	4: ;(*kabinet*)
		IF fb_kl6301_0.GroupReceive.number <10 AND fb_kl6301_0.GroupReceive.number <>0 THEN kabinet_hvac.heat_mode:=fb_kl6301_0.GroupReceive.number;END_IF
		CASE fb_kl6301_0.GroupReceive.number OF
			0:		fb_temp_read(Group_Address:=kabinet_T_EIB_addr, strData_Rec:=fb_KL6301_0.str_Data_Rec, rData=>kabinet_HVAC.cur_t); (*temperature*)
			1:		fb_setpoint_read(Group_address:=kabinet_cooling_EIB_addr, strData_Rec:=fb_KL6301_0.str_Data_Rec, byData=>setpoint_kabinet_dpt4 ); (*cooling*)
					CASE REAL_TO_INT(setpoint_kabinet_dpt4*100/255.0) OF
						0..30:		kabinet_hvac.heat_speed:=1;
									kabinet_hvac.t_ust_cool:= REAL_TO_INT(setpoint_kabinet_dpt4*100/255.0); (*low speed*)
						31..59:		kabinet_hvac.heat_speed:=2;
									kabinet_hvac.t_ust_cool:= REAL_TO_INT(setpoint_kabinet_dpt4*100/255.0-30); (*med speed*)
						60..100:	kabinet_hvac.heat_speed:=3;
									kabinet_hvac.t_ust_cool:= REAL_TO_INT(setpoint_kabinet_dpt4*100/255.0-60); (*high speed*)
					END_CASE
					kabinet_hvac.cur_t_ust:=kabinet_hvac.t_ust_cool;
					(*fb_actual_setpoint_send(group_address:=kabinet_actual_setpoint_addr, str_Rec:=fb_kl6301_0.str_Data_Rec, rData:=kabinet_hvac.cur_t_ust);*)

			2:		fb_setpoint_read(Group_address:=kabinet_heating_EIB_addr, strData_Rec:=fb_KL6301_0.str_Data_Rec, byData=>setpoint_kabinet_dpt4 );  (*heating*)
					CASE REAL_TO_INT(setpoint_kabinet_dpt4*100/255.0) OF
						0..30:		kabinet_hvac.heat_speed:=1;
									kabinet_hvac.t_ust_heat:= REAL_TO_INT(setpoint_kabinet_dpt4*100/255.0); (*low speed*)
						31..59:		kabinet_hvac.heat_speed:=2;
									kabinet_hvac.t_ust_heat:= REAL_TO_INT(setpoint_kabinet_dpt4*100/255.0-30); (*med speed*)
						60..100:	kabinet_hvac.heat_speed:=3;
									kabinet_hvac.t_ust_heat:= REAL_TO_INT(setpoint_kabinet_dpt4*100/255.0-60); (*high speed*)
					END_CASE
					kabinet_hvac.cur_t_ust:=kabinet_hvac.t_ust_heat;
					(*fb_actual_setpoint_send(group_address:=kabinet_actual_setpoint_addr, str_Rec:=fb_kl6301_0.str_Data_Rec, rData:=kabinet_hvac.cur_t_ust);*)


			3:		fb_setpoint_read(Group_address:=kabinet_fan_EIB_addr, strData_Rec:=fb_KL6301_0.str_Data_Rec, byData=>fanspeed_dpt4);
					kabinet_HVAC.heat_speed:=REAL_TO_USINT(fanspeed_dpt4*100/255.0);
			4:		KABINET_HVAC.heat_mode:=0;
			5:		fb_actual_setpoint_read(Group_Address:=kabinet_actual_setpoint_addr, strData_Rec:=fb_KL6301_0.str_Data_Rec );
					kabinet_hvac.cur_t_ust:=fb_actual_setpoint_read.rData;

		END_CASE;

	5: ;(*dytjacha*)
		IF fb_kl6301_0.GroupReceive.number <10 AND fb_kl6301_0.GroupReceive.number <>0 THEN dytjacha_hvac.heat_mode:=fb_kl6301_0.GroupReceive.number;END_IF
		CASE fb_kl6301_0.GroupReceive.number OF
			0:		fb_temp_read(Group_Address:=dytjacha_T_EIB_addr, strData_Rec:=fb_KL6301_0.str_Data_Rec, rData=>dytjacha_HVAC.cur_t); (*temperature*)
			1:		fb_setpoint_read(Group_address:=dytjacha_cooling_EIB_addr, strData_Rec:=fb_KL6301_0.str_Data_Rec, byData=>setpoint_dytjacha_dpt4 ); (*cooling*)
					CASE REAL_TO_INT(setpoint_dytjacha_dpt4*100/255.0) OF
						0..30:		dytjacha_hvac.heat_speed:=1;
									dytjacha_hvac.t_ust_cool:= REAL_TO_INT(setpoint_dytjacha_dpt4*100/255.0); (*low speed*)
						31..59:		dytjacha_hvac.heat_speed:=2;
									dytjacha_hvac.t_ust_cool:= REAL_TO_INT(setpoint_dytjacha_dpt4*100/255.0-30); (*med speed*)
						60..100:	dytjacha_hvac.heat_speed:=3;
									dytjacha_hvac.t_ust_cool:= REAL_TO_INT(setpoint_dytjacha_dpt4*100/255.0-60); (*high speed*)
					END_CASE
					dytjacha_hvac.cur_t_ust:=dytjacha_hvac.t_ust_cool;
					(*fb_actual_setpoint_send(group_address:=dytjacha_actual_setpoint_addr, str_Rec:=fb_kl6301_0.str_Data_Rec, rData:=dytjacha_hvac.cur_t_ust);*)

			2:		fb_setpoint_read(Group_address:=dytjacha_heating_EIB_addr, strData_Rec:=fb_KL6301_0.str_Data_Rec, byData=>setpoint_dytjacha_dpt4 );  (*heating*)
					CASE REAL_TO_INT(setpoint_dytjacha_dpt4*100/255.0) OF
						0..30:		dytjacha_hvac.heat_speed:=1;
									dytjacha_hvac.t_ust_heat:= REAL_TO_INT(setpoint_dytjacha_dpt4*100/255.0); (*low speed*)
						31..59:		dytjacha_hvac.heat_speed:=2;
									dytjacha_hvac.t_ust_heat:= REAL_TO_INT(setpoint_dytjacha_dpt4*100/255.0-30); (*med speed*)
						60..100:	dytjacha_hvac.heat_speed:=3;
									dytjacha_hvac.t_ust_heat:= REAL_TO_INT(setpoint_dytjacha_dpt4*100/255.0-60); (*high speed*)
					END_CASE
					dytjacha_hvac.cur_t_ust:=dytjacha_hvac.t_ust_heat;
					(*fb_actual_setpoint_send(group_address:=dytjacha_actual_setpoint_addr, str_Rec:=fb_kl6301_0.str_Data_Rec, rData:=dytjacha_hvac.cur_t_ust);*)


			3:		fb_setpoint_read(Group_address:=dytjacha_fan_EIB_addr, strData_Rec:=fb_KL6301_0.str_Data_Rec, byData=>fanspeed_dpt4);
					dytjacha_HVAC.heat_speed:=REAL_TO_USINT(fanspeed_dpt4*100/255.0);
			4:		DYTJACHA_HVAC.heat_mode:=0;
			5:		fb_actual_setpoint_read(Group_Address:=dytjacha_actual_setpoint_addr, strData_Rec:=fb_KL6301_0.str_Data_Rec );
					dytjacha_hvac.cur_t_ust:=fb_actual_setpoint_read.rData;

		END_CASE;

	6: ;(*spalnya*)
		IF fb_kl6301_0.GroupReceive.number <10 AND fb_kl6301_0.GroupReceive.number <>0 THEN spalnya_hvac.heat_mode:=fb_kl6301_0.GroupReceive.number;END_IF
		CASE fb_kl6301_0.GroupReceive.number OF
			0:		fb_temp_read(Group_Address:=spalnya_T_EIB_addr, strData_Rec:=fb_KL6301_0.str_Data_Rec, rData=>spalnya_HVAC.cur_t); (*temperature*)
			1:		fb_setpoint_read(Group_address:=spalnya_cooling_EIB_addr, strData_Rec:=fb_KL6301_0.str_Data_Rec, byData=>setpoint_spalnya_dpt4 ); (*cooling*)
					CASE REAL_TO_INT(setpoint_spalnya_dpt4*100/255.0) OF
						0..30:		spalnya_hvac.heat_speed:=1;
									spalnya_hvac.t_ust_cool:= REAL_TO_INT(setpoint_spalnya_dpt4*100/255.0); (*low speed*)
						31..59:		spalnya_hvac.heat_speed:=2;
									spalnya_hvac.t_ust_cool:= REAL_TO_INT(setpoint_spalnya_dpt4*100/255.0-30); (*med speed*)
						60..100:	spalnya_hvac.heat_speed:=3;
									spalnya_hvac.t_ust_cool:= REAL_TO_INT(setpoint_spalnya_dpt4*100/255.0-60); (*high speed*)
					END_CASE
					spalnya_hvac.cur_t_ust:=spalnya_hvac.t_ust_cool;
					(*fb_actual_setpoint_send(group_address:=spalnya_actual_setpoint_addr, str_Rec:=fb_kl6301_0.str_Data_Rec, rData:=spalnya_hvac.cur_t_ust);*)

			2:		fb_setpoint_read(Group_address:=spalnya_heating_EIB_addr, strData_Rec:=fb_KL6301_0.str_Data_Rec, byData=>setpoint_spalnya_dpt4 );  (*heating*)
					CASE REAL_TO_INT(setpoint_spalnya_dpt4*100/255.0) OF
						0..30:		spalnya_hvac.heat_speed:=1;
									spalnya_hvac.t_ust_heat:= REAL_TO_INT(setpoint_spalnya_dpt4*100/255.0); (*low speed*)
						31..59:		spalnya_hvac.heat_speed:=2;
									spalnya_hvac.t_ust_heat:= REAL_TO_INT(setpoint_spalnya_dpt4*100/255.0-30); (*med speed*)
						60..100:	spalnya_hvac.heat_speed:=3;
									spalnya_hvac.t_ust_heat:= REAL_TO_INT(setpoint_spalnya_dpt4*100/255.0-60); (*high speed*)
					END_CASE
					spalnya_hvac.cur_t_ust:=spalnya_hvac.t_ust_heat;
					(*fb_actual_setpoint_send(group_address:=spalnya_actual_setpoint_addr, str_Rec:=fb_kl6301_0.str_Data_Rec, rData:=spalnya_hvac.cur_t_ust);*)


			3:		fb_setpoint_read(Group_address:=spalnya_fan_EIB_addr, strData_Rec:=fb_KL6301_0.str_Data_Rec, byData=>fanspeed_dpt4);
					spalnya_HVAC.heat_speed:=REAL_TO_USINT(fanspeed_dpt4*100/255.0);
			4:		SPALNYA_HVAC.heat_mode:=0;
			5:		fb_actual_setpoint_read(Group_Address:=spalnya_actual_setpoint_addr, strData_Rec:=fb_KL6301_0.str_Data_Rec );
					spalnya_hvac.cur_t_ust:=fb_actual_setpoint_read.rData;

		END_CASE;
END_CASE



(*hdl gate can transmit 2byte values, but they can not be assigned to DLP panel AC unit setpoint value directly,
so for every setpoint value in range [20,30] a 1 bit eib telegram with corresponding  adress +100 ( [120,130] ) should be generated and transmitted to HDL logic module and then
logic module assigns it to apropriate value DLP panel AC unit. 
amen*)
fb_setpoint_switch_send.iMode:=2;
fb_setpoint_switch_send.bStart:=TRUE;
IF vitalnya_hvac.cur_t_ust_prev <> vitalnya_hvac.cur_t_ust THEN
	fb_setpoint_switch_send.Group_Address.NUMBER:=REAL_TO_BYTE(vitalnya_hvac.cur_t_ust)+100;
	fb_setpoint_switch_send.Group_Address.MAIN:=1;
	fb_setpoint_switch_send.Group_Address.SUB_MAIN:=1;
	fb_setpoint_switch_send(str_Rec:=fb_KL6301_0.str_Data_Rec, bData:=FALSE);
	fb_setpoint_switch_send(str_Rec:=fb_KL6301_0.str_Data_Rec, bData:=TRUE);
END_IF
IF kino_hvac.cur_t_ust_prev <> kino_hvac.cur_t_ust THEN
	fb_setpoint_switch_send.Group_Address.NUMBER:=REAL_TO_BYTE(kino_hvac.cur_t_ust)+100;
	fb_setpoint_switch_send.Group_Address.MAIN:=1;
	fb_setpoint_switch_send.Group_Address.SUB_MAIN:=2;
	fb_setpoint_switch_send(str_Rec:=fb_KL6301_0.str_Data_Rec, bData:=1);
	fb_setpoint_switch_send(str_Rec:=fb_KL6301_0.str_Data_Rec, bData:=0);
END_IF
IF studio_hvac.cur_t_ust_prev <> studio_hvac.cur_t_ust THEN
	fb_setpoint_switch_send.Group_Address.NUMBER:=REAL_TO_BYTE(studio_hvac.cur_t_ust)+100;
	fb_setpoint_switch_send.Group_Address.MAIN:=1;
	fb_setpoint_switch_send.Group_Address.SUB_MAIN:=3;
	fb_setpoint_switch_send(str_Rec:=fb_KL6301_0.str_Data_Rec, bData:=1);
	fb_setpoint_switch_send(str_Rec:=fb_KL6301_0.str_Data_Rec, bData:=0);
END_IF
IF kabinet_hvac.cur_t_ust_prev <> kabinet_hvac.cur_t_ust THEN
	fb_setpoint_switch_send.Group_Address.NUMBER:=REAL_TO_BYTE(kabinet_hvac.cur_t_ust)+100;
	fb_setpoint_switch_send.Group_Address.MAIN:=1;
	fb_setpoint_switch_send.Group_Address.SUB_MAIN:=4;
	fb_setpoint_switch_send(str_Rec:=fb_KL6301_0.str_Data_Rec, bData:=1);
	fb_setpoint_switch_send(str_Rec:=fb_KL6301_0.str_Data_Rec, bData:=0);
END_IF
IF dytjacha_hvac.cur_t_ust_prev <> dytjacha_hvac.cur_t_ust THEN
	fb_setpoint_switch_send.Group_Address.NUMBER:=REAL_TO_BYTE(dytjacha_hvac.cur_t_ust)+100;
	fb_setpoint_switch_send.Group_Address.MAIN:=1;
	fb_setpoint_switch_send.Group_Address.SUB_MAIN:=5;
	fb_setpoint_switch_send(str_Rec:=fb_KL6301_0.str_Data_Rec, bData:=1);
	fb_setpoint_switch_send(str_Rec:=fb_KL6301_0.str_Data_Rec, bData:=0);
END_IF
IF spalnya_hvac.cur_t_ust_prev <> spalnya_hvac.cur_t_ust THEN
	fb_setpoint_switch_send.Group_Address.NUMBER:=REAL_TO_BYTE(spalnya_hvac.cur_t_ust)+100;
	fb_setpoint_switch_send.Group_Address.MAIN:=1;
	fb_setpoint_switch_send.Group_Address.SUB_MAIN:=6;
	fb_setpoint_switch_send(str_Rec:=fb_KL6301_0.str_Data_Rec, bData:=1);
	fb_setpoint_switch_send(str_Rec:=fb_KL6301_0.str_Data_Rec, bData:=0);
END_IF
END_ACTION
ACTION timers:
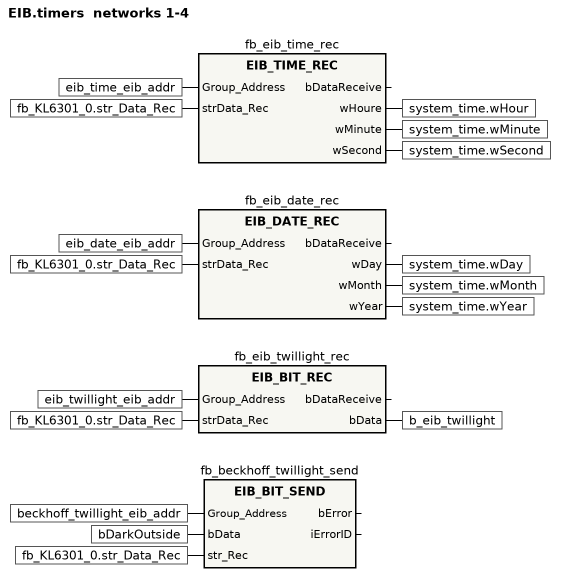
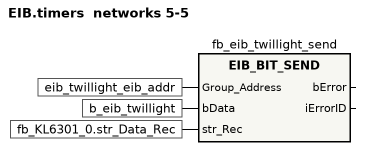
_FBD_ (* Function Block Diagram *)
NETWORK 1
	fb_eib_time_rec:EIB_TIME_REC(Group_Address: eib_time_eib_addr, strData_Rec: fb_KL6301_0.str_Data_Rec, wHoure => system_time.wHour, wMinute => system_time.wMinute, wSecond => system_time.wSecond)
NETWORK 2
	fb_eib_date_rec:EIB_DATE_REC(Group_Address: eib_date_eib_addr, strData_Rec: fb_KL6301_0.str_Data_Rec, wDay => system_time.wDay, wMonth => system_time.wMonth, wYear => system_time.wYear)
NETWORK 3
	fb_eib_twillight_rec:EIB_BIT_REC(Group_Address: eib_twillight_eib_addr, strData_Rec: fb_KL6301_0.str_Data_Rec, bData => b_eib_twillight)
NETWORK 4
	fb_beckhoff_twillight_send:EIB_BIT_SEND(Group_Address: beckhoff_twillight_eib_addr, bData: bDarkOutside, str_Rec: fb_KL6301_0.str_Data_Rec)
NETWORK 5
	fb_eib_twillight_send:EIB_BIT_SEND(Group_Address: eib_twillight_eib_addr, bData: b_eib_twillight, str_Rec: fb_KL6301_0.str_Data_Rec)
_END_FBD_
(* the same logic as Structured Text *)
(* Network 1 *)
fb_eib_time_rec(Group_Address := eib_time_eib_addr, strData_Rec := fb_KL6301_0.str_Data_Rec);
system_time.wHour := fb_eib_time_rec.wHoure;
system_time.wMinute := fb_eib_time_rec.wMinute;
system_time.wSecond := fb_eib_time_rec.wSecond;
(* Network 2 *)
fb_eib_date_rec(Group_Address := eib_date_eib_addr, strData_Rec := fb_KL6301_0.str_Data_Rec);
system_time.wDay := fb_eib_date_rec.wDay;
system_time.wMonth := fb_eib_date_rec.wMonth;
system_time.wYear := fb_eib_date_rec.wYear;
(* Network 3 *)
fb_eib_twillight_rec(Group_Address := eib_twillight_eib_addr, strData_Rec := fb_KL6301_0.str_Data_Rec);
b_eib_twillight := fb_eib_twillight_rec.bData;
(* Network 4 *)
fb_beckhoff_twillight_send(Group_Address := beckhoff_twillight_eib_addr, bData := bDarkOutside, str_Rec := fb_KL6301_0.str_Data_Rec);
(* Network 5 *)
fb_eib_twillight_send(Group_Address := eib_twillight_eib_addr, bData := b_eib_twillight, str_Rec := fb_KL6301_0.str_Data_Rec);
END_ACTION

(* POU RANGE_TO_RANGE, ST *)
FUNCTION RANGE_TO_RANGE : INT
VAR_INPUT
	by_input:BYTE;
	in_low_value: INT;
	in_high_value:INT;
	out_low_value: INT;
	out_high_value:INT;
END_VAR
VAR
	r_res: REAL;
	r_input: REAL;
END_VAR
r_input:=BYTE_TO_REAL(by_input);
IF out_high_value>out_low_value THEN
	r_res:=r_input/(in_high_value - in_low_value)*(out_high_value - out_low_value);
ELSE
	r_res:=out_low_value - (r_input / (in_high_value - in_low_value)*(out_low_value - out_high_value));
END_IF
RANGE_TO_RANGE:=REAL_TO_INT(r_res);
END_FUNCTION

(* POU GREATEST_OF, ST *)
FUNCTION GREATEST_OF : REAL
VAR_INPUT
	r_in1,r_in2:REAL;
END_VAR
VAR
END_VAR
IF r_in1>=r_in2 THEN
	GREATEST_OF:=r_in1;
ELSE
	GREATEST_OF:=r_in2;
END_IF
END_FUNCTION

(* POU LIGHT, ST *)
PROGRAM LIGHT
VAR
	tambur1, tambur2,tambur3 : SWITCH;
	korydor : SWITCH;
	spalnya1,spalnya2, spalnya_balk:SWITCH;
	dytjacha1,dytjacha2  : SWITCH;
	su1 : SWITCH;
	su2: SWITCH;
	garderob1, garderob2 : SWITCH;

	tLightWindow: TIME;		(*Час, який світло світиться після спрацювання сенсора руху*)

	VENT_TIMER: TOF;		(*Таймер роботи вентилятора в пустому туалеті*)
	vent_timer_start: R_TRIG;
	test: BOOL;

	CHOVEN_TIMER: TOF;	(*Таймер роботи світильника на човні*)

	bChovenTimerOverride: SEMA;		(*Перевага вимикача над таймером*)
	bGarderobTimerOverride: SEMA;		(*Перевага вимикача над таймером*)
	KORYDOR_TIMER: TOF;		(*Таймер роботи світла в коридорі*)
	KORYDOR_F: F_TRIG;
	GARDEROB_TIMER: TOF;		(*Таймер роботи світла в гардеробі*)
	GARDEROB_F: F_TRIG;		(*Спрацювання сенсора руху в гардеробі*)
	KORYDOR_SEMA:SEMA;
	su_light: BOOL;
	vymykach3: BOOL;

	fb_light_write:EIB_BIT_SEND;
	block_korydor, block_garderob, block_choven: BOOL;

END_VAR
tLightWindow:=t#60s;

IF fb_moove_sensors_read.bData THEN
	moove_sensors:=(*bDarkOutside*)TRUE;
ELSE
	moove_sensors:=FALSE;
END_IF

(*Опитування вимикачів*)
tambur1(IN:=sw_tambur1);
tambur2(IN:=sw_tambur3_2);
tambur3(IN:=sw_tambur3);



spalnya1(IN:=sw_spalnya1 XOR sw_spalnya4);
spalnya2(IN:=sw_spalnya2 XOR sw_spalnya3);
spalnya_balk(IN:=sw_spalnya_balk);

dytjacha1(IN:=sw_dytjacha1);
dytjacha2(IN:=sw_dytjacha2);

su1(IN:=sw_su1);
su2(IN:=sw_su2);




(*запуск вечірніх таймерів світла*)





(*обробка сигналів вимикачів та таймерів*)
IF fb_bar_read.bDataReceive THEN
	IF tambur1.short THEN bar:= NOT bar; END_IF
ELSE
	bar:=fb_bar_read.bData;
END_IF

(*Відправка на 1,2 поверхи значення вимикача*)
data2floor[6].0:=sw_tambur3_2;
data1floor[2].1:=sw_tambur3_2;

CHOVEN_TIMER(IN:= NOT fb_choven_read.bData AND NOT moove_skhody, PT:= tLightWindow);
IF fb_choven_read.bData THEN
	choven:=TRUE;
ELSE
	IF moove_sensors  AND  CHOVEN_timer.Q	THEN  choven:=TRUE;
	ELSE
	choven:=FALSE;
	END_IF
END_IF


korydor(IN:=sw_korydor);
KORYDOR_TIMER(IN:=  NOT fb_korydor_lampa_read.bData  AND NOT moove_korydor, PT:= tLightWindow);

IF fb_korydor_lampa_read.bData THEN
	korydor_lampa:=TRUE;
ELSE
		korydor_lampa:=KORYDOR_TIMER.Q;
END_IF

IF fb_korydor_skeli_read.bData THEN
	korydor_skeli:=TRUE;
ELSE
	korydor_skeli:=KORYDOR_TIMER.Q;
END_IF

IF fb_korydor_svitlo_read.bDataReceive THEN
	KORYDOR_F(clk:=korydor_timer.Q);
	KORYDOR_SEMA(CLAIM:=(NOT korydor_svitlo AND korydor.short ), RELEASE:=(korydor_svitlo AND korydor.short) OR KORYDOR_f.Q);
	korydor_svitlo:=KORYDOR_SEMA.BUSY;
ELSE
	korydor_svitlo:= fb_korydor_svitlo_read.bData;

END_IF

IF fb_spalnya_kulbaba_read.bDataReceive THEN
	IF spalnya1.short THEN spalnya_kulbaba:=NOT spalnya_kulbaba; END_IF
ELSE
	spalnya_kulbaba:=fb_spalnya_kulbaba_read.bData;
END_IF

IF fb_spalnya_kontrazhur_read.bDataReceive XOR fb_spalnya_kontrazhur_b_read.bDataReceive  XOR fb_spalnya_kontrazhur_l_read.bDataReceive  THEN
	IF spalnya2.short THEN
		 spalnya_kontrazhur:= NOT spalnya_kontrazhur;
		spalnya_kontrazhur_b:=spalnya_kontrazhur;
		spalnya_kontrazhur_l:=spalnya_kontrazhur;
 	END_IF
ELSE
	IF NOT fb_spalnya_kontrazhur_read.bDataReceive THEN spalnya_kontrazhur:= fb_spalnya_kontrazhur_read.bData; END_IF
	IF NOT fb_spalnya_kontrazhur_l_read.bDataReceive THEN spalnya_kontrazhur_l:= fb_spalnya_kontrazhur_l_read.bData; END_IF
	IF NOT fb_spalnya_kontrazhur_b_read.bDataReceive THEN spalnya_kontrazhur_b:= fb_spalnya_kontrazhur_b_read.bData; END_IF
END_IF

IF fb_spalnya_balkon_read.bDataReceive THEN
	IF  spalnya_balk.short  THEN spalnya_balkon:=NOT spalnya_balkon; END_IF
ELSE
	spalnya_balkon:=fb_spalnya_balkon_read.bData;
END_IF

IF fb_dytjacha_read.bDataReceive THEN
	IF dytjacha1.short THEN dytjacha:= NOT dytjacha; END_IF
ELSE
	dytjacha:=fb_dytjacha_read.bData;
END_IF

IF fb_dytjacha_bra_read.bDataReceive THEN
	IF dytjacha2.short THEN dytjacha_bra:= NOT dytjacha_bra; END_IF
ELSE
	dytjacha_bra:=fb_dytjacha_bra_read.bData;
END_IF


IF fb_su3_stina_read.bDataReceive AND  fb_su3_kontrazhur_k_read.bDataReceive THEN
	IF su2.short THEN
		su3_stina:= NOT su3_stina;
		(*su3_kontrazhur_k:= su3_stina; *)
	END_IF
ELSE
	IF NOT fb_su3_stina_read.bDataReceive THEN
		 su3_stina:=fb_su3_stina_read.bData;
	END_IF
	IF NOT fb_su3_kontrazhur_k_read.bDataReceive THEN
		su3_kontrazhur_k:= fb_su3_kontrazhur_k_read.bData;
	END_IF
END_IF



IF fb_su3_bra_read.bDataReceive XOR fb_su3_lampa_read.bDataReceive XOR fb_su3_kontrazhur_read.bDataReceive THEN
	IF su2.long THEN
		su3_bra:= NOT su3_bra;
		su3_lampa:= su3_bra;
		su3_kontrazhur:=su3_lampa;
	END_IF
ELSE
	IF NOT  fb_su3_bra_read.bDataReceive THEN su3_bra:= fb_su3_bra_read.bData;END_IF
	IF NOT fb_su3_lampa_read.bDataReceive THEN su3_lampa:=fb_su3_lampa_read.bData; END_IF
	IF NOT  fb_su3_kontrazhur_read.bDataReceive THEN su3_kontrazhur:=fb_su3_kontrazhur_read.bData; END_IF
END_IF

IF su1.long THEN su3_vent:= NOT su3_vent; END_IF

IF fb_su3_pidsvitka_read.bDataReceive THEN
	IF su1.short THEN su3_pidsvitka:= NOT su3_pidsvitka; END_IF
ELSE
	su3_pidsvitka:=fb_su3_pidsvitka_read.bData;
END_IF

(*IF su1.short AND NOT su3_vent THEN su3_vent:=TRUE; END_IF; *) (*вмикання вентилятора разом зі світлом*)

(*
вмикання вентилятора на деякий час після того, як вимикається все світло у ванній

su_light:=su3_stina OR su3_kontrazhur OR su3_bra OR su3_pidsvitka;

vent_timer_start(CLK:=NOT su_light );
VENT_TIMER(PT:=tOffDelay,IN:=vent_timer_start.Q);
IF NOT su_light THEN
	su3_vent:= VENT_TIMER.Q;
END_IF
*)


garderob1(IN:=sw_garderob1);
garderob2(IN:=sw_garderob2);
GARDEROB_F(CLK:=moove_garderob);
GARDEROB_TIMER(IN:= GARDEROB_F.Q, PT:= tLightWindow*2);

IF fb_serverna_read.bDataReceive THEN
	IF garderob2.short THEN serverna := NOT serverna; END_IF
ELSE
	Serverna:=fb_serverna_read.bData;
END_IF

IF fb_garderob_read.bDataReceive THEN
(*	bGarderobTimerOverride(CLAIM:=  (NOT moove_garderob OR (NOT garderob AND garderob1.short)), RELEASE:=  (garderob AND  garderob1.short) );
	garderob:=bGarderobTimerOverride.BUSY;*)
	IF garderob1.short THEN garderob:= NOT garderob; END_IF
ELSE
	garderob:=fb_garderob_read.bData;
END_IF
END_PROGRAM

(* POU Vymykachi/SWITCH, ST *)
FUNCTION_BLOCK SWITCH
VAR_INPUT
	IN:BOOL;
	SHORT_OFF_DELAY, LONG_OFF_DELAY: TIME; (*час затримки вимкнення по короткому та довгому натисненню*)
END_VAR
VAR_OUTPUT
	short, long:BOOL;
END_VAR
VAR
	tChas: TIME; (*час доки кнопка натиснена*)
	TIMER: TON; (*таймер час натискання*)
	bPressed:BOOL;
	turn_off_long: BOOL;
	start_l, start_s:BOOL;
	bStan: BOOL:=FALSE;
END_VAR
short:=FALSE;
long:=FALSE;
TIMER(IN:=IN AND bStan, PT:=t#10s);
IF IN AND bStan THEN
	tChas:=timer.ET;
	bPressed:=TRUE;
ELSE
	bPressed:=FALSE;
END_IF;

IF NOT IN AND NOT bStan THEN
	tChas:=t#0ms;
END_IF;

IF bStan AND NOT IN THEN
	IF tChas <tLongPress THEN
		short:=TRUE;
	END_IF;
	IF tChas>=tLongPress THEN
		long:=TRUE;
	END_IF;
END_IF;
bStan := IN;
END_FUNCTION_BLOCK

(* POU shtory, ST *)
PROGRAM shtory
VAR
	inc1, inc: UINT;
	impulse: BOOL;
	last_move: UINT;
	impulse1: BOOL;
	last_move1: UINT;
	lift_move_dir, lift_move: BOOL;
	rising1: BOOL;
	falling1: BOOL;
	rising2: BOOL;
	falling2: BOOL;
	panel_shtory_move, panel_tul_move, panel_lift_move:BOOL;

	(*таймери для формування керуючих імпульсів*)
	timer_shtory_move, timer_shtory_stop,timer_tul_move, timer_tul_stop, move_lift_up, move_lift_down: TP;
	counter:CTU;
	shtory_move: BOOL;
	tul_move: BOOL;
	bBlock:BOOL;
	darkness_shtory_move: TP;
	btest: BOOL;

	eib_spalnya_shtory_status_send: EIB_BIT_SEND;
	eib_spalnya_tul_status_send: EIB_BIT_SEND;
	spalnya_shtory_status: BOOL;
	spalnya_tul_status: BOOL;
END_VAR
bBlock:=FALSE;
IF MAIN.fbRTC.stSystemTime.wHour=11 AND MAIN.fbRTC.stSystemTime.wMinute=0 AND MAIN.fbRTC.stSystemTime.wSecond<22 THEN
	bBlock:=TRUE;
	lift_down:=TRUE;
	lift_up:=FALSE;
	lift_move_dir:=FALSE;
	shtory_open:=TRUE;
	shtory_close:=FALSE;
	tul_open:=FALSE;
	tul_close:=TRUE;

ELSE
	(*детекція відсутності фронтів*)
	IF LIGHT.spalnya1.long = impulse THEN
		rising1:=0;
		falling1:=0;
	END_IF;

	IF LIGHT.spalnya2.long = impulse1  THEN
		rising2:=0;
		falling2:=0;
	END_IF;

	(*якщо клавіші довго  натиснені одночасно, то рухати ліфт, якщо довго і окремо - штори*)
	IF ( (LIGHT.spalnya1.long AND LIGHT.spalnya2.long) OR panel_lift_move)  AND NOT( move_lift_up.Q OR  move_lift_down.Q)  THEN
		lift_move:=1;
		lift_move_dir:= NOT lift_move_dir;
	ELSE

		(*ловим передній фронт довгого натискання першої клавіші*)
		IF LIGHT.spalnya1.long AND NOT impulse  AND NOT LIGHT.spalnya2.long THEN
			rising1:=1;
			falling1:=0;
		END_IF;

		(*задній фронт*)
		IF NOT LIGHT.spalnya1.long AND  impulse AND NOT LIGHT.spalnya2.long  THEN
			falling1:=1;
			rising1:=0;
		END_IF;

		(*ловим передній фронт довгого натискання другої клавіші*)
		IF LIGHT.spalnya2.long AND NOT impulse1 AND NOT LIGHT.spalnya1.long  THEN
			rising2:=1;
			falling2:=0;
		END_IF;

		(*ловим задній фронт довгого натискання другої клавіші*)
		IF NOT LIGHT.spalnya2.long AND  impulse1 AND NOT LIGHT.spalnya1.long THEN
			falling2:=1;
			rising2:=0;
		END_IF
	END_IF
	(*команди шторам та ліфту з панелей смартбаса*)
	eib_shtory(Group_Address:=shtory_spalnya_EIB_addr, strData_Rec:=fb_KL6301_0.str_Data_Rec);
	eib_tul(Group_Address:=tul_spalnya_EIB_addr, strData_Rec:=fb_KL6301_0.str_Data_Rec);
	eib_lift(Group_Address:=lift_spalnya_EIB_addr, strData_Rec:=fb_KL6301_0.str_Data_Rec);


	IF NOT eib_shtory_kabinet.bDataReceive THEN data2floor[7].0:=eib_shtory_kabinet.bData; END_IF
	IF NOT eib_tul_kabinet.bDataReceive THEN data2floor[7].1:=eib_tul_kabinet.bData; END_IF
	IF NOT eib_shtory_kino.bDataReceive THEN data2floor[7].2:=eib_shtory_kino.bData; END_IF
	IF NOT eib_tul_kino.bDataReceive THEN data2floor[7].3:=eib_tul_kino.bData; END_IF

	panel_tul_move:= NOT eib_tul.bDataReceive;
	panel_shtory_move:= NOT eib_shtory.bDataReceive;
	panel_lift_move:=NOT eib_lift.bDataReceive;


	shtory_move:= LIGHT.spalnya1.long OR panel_shtory_move;
	tul_move:= LIGHT.spalnya2.long OR panel_tul_move;



	(*формування імпульсів для керування шторами, тюлями та ліфтом*)
	timer_shtory_move(IN:=shtory_move, PT:=t#500ms);
	timer_shtory_stop(IN:=shtory_move , PT:=t#500ms);
	timer_tul_move(IN:=tul_move  , PT:=t#500ms);
	timer_tul_stop(IN:=tul_move , PT:=t#500ms);

	move_lift_up(IN:=lift_move AND lift_move_dir , PT:=t#20s,Q=>lift_up);
	move_lift_down(IN:=lift_move AND NOT lift_move_dir, PT:=t#20s, Q=>lift_down);



	darkness_shtory_move(IN:=bDarkOutside, PT:=t#15s);
	IF darkness_shtory_move.Q THEN
		shtory_open:=FALSE;
		shtory_close:=TRUE;
		tul_open:=FALSE;
		tul_close:=TRUE;
		bBlock:=TRUE;
	END_IF


	IF NOT bBlock THEN
		IF NOT (LIGHT.spalnya1.long AND LIGHT.spalnya2.long) THEN (*якщо не засік довгого затискання двох клавіш (ліфт не рухається) - рухати штори *)

		(*вибір рухати чи зупинити  штори*)
			IF shtory_move   THEN
				inc:=inc+1;
			END_IF;
			IF inc>2 THEN inc:=1; END_IF;

			(*вибір рухати чи зупинити  тюль*)
			IF tul_move THEN
				inc1:=inc1+1;
			END_IF;
			IF inc1>2 THEN inc1:=1; END_IF;

			CASE inc OF

				1:
				shtory_open:=timer_shtory_move.Q; (*відкривати*)
				shtory_close:= 0;
				last_move:=inc;
				spalnya_shtory_status:=1;

				2:
				shtory_close:=timer_shtory_move.Q;(*закривати*)
				shtory_open:= 0;
				last_move:=inc;
				spalnya_shtory_status:=0;

			END_CASE;

			CASE inc1 OF

				1:
				tul_open:=timer_tul_move.Q; (*відкривати*)
				tul_close:= 0;
				last_move1:=inc;
				spalnya_tul_status:=1;
				2:
				tul_close:=timer_tul_move.Q;(*закривати*)
				tul_open:= 0;
				last_move1:=inc;
				spalnya_tul_status:=0;
			END_CASE;

		END_IF;
	END_IF

	(*запам'ятовування стану довгого натискання для детекції фронтів*)

	impulse:=LIGHT.spalnya1.long;
	impulse1:=LIGHT.spalnya2.long;

	 lift_move:= 0;
END_IF
eib_status_send;

new_shtory;
END_PROGRAM
ACTION eib_status_send:
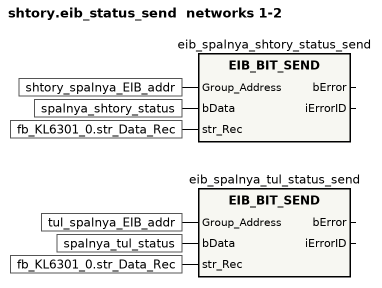
_FBD_ (* Function Block Diagram *)
NETWORK 1
	eib_spalnya_shtory_status_send:EIB_BIT_SEND(Group_Address: shtory_spalnya_EIB_addr, bData: spalnya_shtory_status, str_Rec: fb_KL6301_0.str_Data_Rec)
NETWORK 2
	eib_spalnya_tul_status_send:EIB_BIT_SEND(Group_Address: tul_spalnya_EIB_addr, bData: spalnya_tul_status, str_Rec: fb_KL6301_0.str_Data_Rec)
_END_FBD_
(* the same logic as Structured Text *)
(* Network 1 *)
eib_spalnya_shtory_status_send(Group_Address := shtory_spalnya_EIB_addr, bData := spalnya_shtory_status, str_Rec := fb_KL6301_0.str_Data_Rec);
(* Network 2 *)
eib_spalnya_tul_status_send(Group_Address := tul_spalnya_EIB_addr, bData := spalnya_tul_status, str_Rec := fb_KL6301_0.str_Data_Rec);
END_ACTION

(* POU new_shtory, CFC *)
PROGRAM new_shtory
VAR

END_VAR
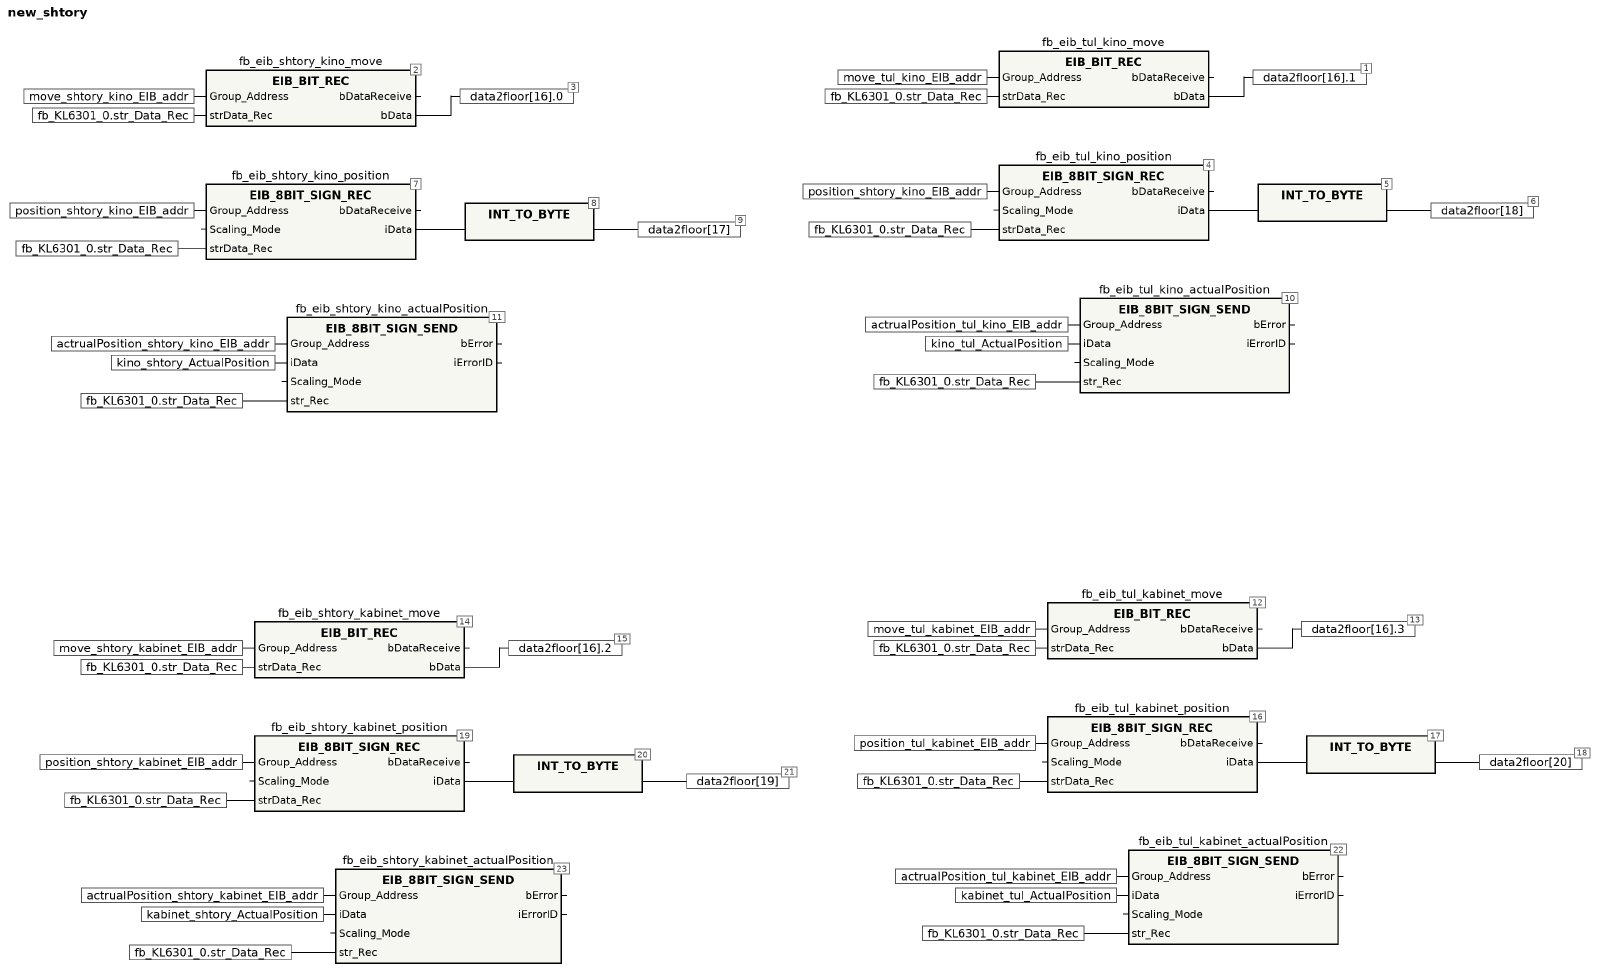
_CFC_ (* Continuous Function Chart, elements in execution order *)
#0 fb_eib_tul_kino_move:EIB_BIT_REC(Group_Address: move_tul_kino_EIB_addr, strData_Rec: fb_KL6301_0.str_Data_Rec)
#1 data2floor[16].1 <= #0.bData
#2 fb_eib_shtory_kino_move:EIB_BIT_REC(Group_Address: move_shtory_kino_EIB_addr, strData_Rec: fb_KL6301_0.str_Data_Rec)
#3 data2floor[16].0 <= #2.bData
#4 fb_eib_tul_kino_position:EIB_8BIT_SIGN_REC(Group_Address: position_shtory_kino_EIB_addr, Scaling_Mode: -, strData_Rec: fb_KL6301_0.str_Data_Rec)
#5 INT_TO_BYTE(#4.iData)
#6 data2floor[18] <= #5
#7 fb_eib_shtory_kino_position:EIB_8BIT_SIGN_REC(Group_Address: position_shtory_kino_EIB_addr, Scaling_Mode: -, strData_Rec: fb_KL6301_0.str_Data_Rec)
#8 INT_TO_BYTE(#7.iData)
#9 data2floor[17] <= #8
#10 fb_eib_tul_kino_actualPosition:EIB_8BIT_SIGN_SEND(Group_Address: actrualPosition_tul_kino_EIB_addr, iData: kino_tul_ActualPosition, Scaling_Mode: -, str_Rec: fb_KL6301_0.str_Data_Rec)
#11 fb_eib_shtory_kino_actualPosition:EIB_8BIT_SIGN_SEND(Group_Address: actrualPosition_shtory_kino_EIB_addr, iData: kino_shtory_ActualPosition, Scaling_Mode: -, str_Rec: fb_KL6301_0.str_Data_Rec)
#12 fb_eib_tul_kabinet_move:EIB_BIT_REC(Group_Address: move_tul_kabinet_EIB_addr, strData_Rec: fb_KL6301_0.str_Data_Rec)
#13 data2floor[16].3 <= #12.bData
#14 fb_eib_shtory_kabinet_move:EIB_BIT_REC(Group_Address: move_shtory_kabinet_EIB_addr, strData_Rec: fb_KL6301_0.str_Data_Rec)
#15 data2floor[16].2 <= #14.bData
#16 fb_eib_tul_kabinet_position:EIB_8BIT_SIGN_REC(Group_Address: position_tul_kabinet_EIB_addr, Scaling_Mode: -, strData_Rec: fb_KL6301_0.str_Data_Rec)
#17 INT_TO_BYTE(#16.iData)
#18 data2floor[20] <= #17
#19 fb_eib_shtory_kabinet_position:EIB_8BIT_SIGN_REC(Group_Address: position_shtory_kabinet_EIB_addr, Scaling_Mode: -, strData_Rec: fb_KL6301_0.str_Data_Rec)
#20 INT_TO_BYTE(#19.iData)
#21 data2floor[19] <= #20
#22 fb_eib_tul_kabinet_actualPosition:EIB_8BIT_SIGN_SEND(Group_Address: actrualPosition_tul_kabinet_EIB_addr, iData: kabinet_tul_ActualPosition, Scaling_Mode: -, str_Rec: fb_KL6301_0.str_Data_Rec)
#23 fb_eib_shtory_kabinet_actualPosition:EIB_8BIT_SIGN_SEND(Group_Address: actrualPosition_shtory_kabinet_EIB_addr, iData: kabinet_shtory_ActualPosition, Scaling_Mode: -, str_Rec: fb_KL6301_0.str_Data_Rec)
_END_CFC_
(* the same logic as Structured Text *)
fb_eib_tul_kino_move(Group_Address := move_tul_kino_EIB_addr, strData_Rec := fb_KL6301_0.str_Data_Rec);
data2floor[16].1 := fb_eib_tul_kino_move.bData;
fb_eib_shtory_kino_move(Group_Address := move_shtory_kino_EIB_addr, strData_Rec := fb_KL6301_0.str_Data_Rec);
data2floor[16].0 := fb_eib_shtory_kino_move.bData;
fb_eib_tul_kino_position(Group_Address := position_shtory_kino_EIB_addr, strData_Rec := fb_KL6301_0.str_Data_Rec);
data2floor[18] := INT_TO_BYTE(fb_eib_tul_kino_position.iData);
fb_eib_shtory_kino_position(Group_Address := position_shtory_kino_EIB_addr, strData_Rec := fb_KL6301_0.str_Data_Rec);
data2floor[17] := INT_TO_BYTE(fb_eib_shtory_kino_position.iData);
fb_eib_tul_kino_actualPosition(Group_Address := actrualPosition_tul_kino_EIB_addr, iData := kino_tul_ActualPosition, str_Rec := fb_KL6301_0.str_Data_Rec);
fb_eib_shtory_kino_actualPosition(Group_Address := actrualPosition_shtory_kino_EIB_addr, iData := kino_shtory_ActualPosition, str_Rec := fb_KL6301_0.str_Data_Rec);
fb_eib_tul_kabinet_move(Group_Address := move_tul_kabinet_EIB_addr, strData_Rec := fb_KL6301_0.str_Data_Rec);
data2floor[16].3 := fb_eib_tul_kabinet_move.bData;
fb_eib_shtory_kabinet_move(Group_Address := move_shtory_kabinet_EIB_addr, strData_Rec := fb_KL6301_0.str_Data_Rec);
data2floor[16].2 := fb_eib_shtory_kabinet_move.bData;
fb_eib_tul_kabinet_position(Group_Address := position_tul_kabinet_EIB_addr, strData_Rec := fb_KL6301_0.str_Data_Rec);
data2floor[20] := INT_TO_BYTE(fb_eib_tul_kabinet_position.iData);
fb_eib_shtory_kabinet_position(Group_Address := position_shtory_kabinet_EIB_addr, strData_Rec := fb_KL6301_0.str_Data_Rec);
data2floor[19] := INT_TO_BYTE(fb_eib_shtory_kabinet_position.iData);
fb_eib_tul_kabinet_actualPosition(Group_Address := actrualPosition_tul_kabinet_EIB_addr, iData := kabinet_tul_ActualPosition, str_Rec := fb_KL6301_0.str_Data_Rec);
fb_eib_shtory_kabinet_actualPosition(Group_Address := actrualPosition_shtory_kabinet_EIB_addr, iData := kabinet_shtory_ActualPosition, str_Rec := fb_KL6301_0.str_Data_Rec);
END_PROGRAM

(* POU HVAC/climate, ST *)
PROGRAM climate
VAR PERSISTENT

	t_out_avg_day, t_out_avg_10day:REAL;
	measures_this_day, meashured_days:INT;
	day_sum, ten_day_sum:REAL;
END_VAR


VAR

	t_tambur: REAL;
	t_su: REAL;
	t_spalnya : REAL;
	(*мінімум та максимум температур теплих підлог*)
	t_max: REAL;
	t_min: REAL;

	i: INT:=0;
	OAT_filter: 			FB_PT1;
	(*sensor filters*)
	t_tambur_filter: 		FB_PT1;
	t_su_filter : 			FB_PT1;
	t_spalnya_filter: 		FB_PT1;

	temperatureFiltersCycleTime:	TIME:=t#28ms;
	temperaturesFilterT1:			TIME:=t#60s;




END_VAR
(*фільтри показань сенсорів температури*)

OAT_filter.tCycletime:=temperatureFiltersCycleTime;
OAT_filter.tT1:=temperaturesFilterT1;
OAT_filter(fIn:=INT_TO_REAL(iT_out)/10, fOut=>t_out);

t_tambur_filter.tCycletime:=temperatureFiltersCycleTime;
t_tambur_filter.tT1:=temperaturesFilterT1;
t_tambur_filter (fIn:=INT_TO_REAL(iT_tambur)/10, fOut=>t_tambur);

t_su_filter.tCycletime:=temperatureFiltersCycleTime;
t_su_filter.tT1:=temperaturesFilterT1;
t_su_filter(fIn:=INT_TO_REAL(iT_su)/10, fOut=>t_su);

t_spalnya_filter.tCycletime:=temperatureFiltersCycleTime;
t_spalnya_filter.tT1:=temperaturesFilterT1;
t_spalnya_filter(fIn:=INT_TO_REAL(iT_spalnya)/10, fOut=>t_spalnya);


(*CASE MAIN.fbRTC.stSystemTime.wSecond OF*)



(*summer; *)

t_max:=70;
t_min:=20;
IF t_out<15 THEN

	IF t_tambur > t_max THEN (*вимкнути колектор, якщо підлога тепліша за верхню межу температури*)
		freshbar_col:=FALSE;
	ELSE
		IF t_tambur< t_min THEN (*увімкнути колектор, якщо підлога холодніша за нижню межу*)
			freshbar_col:=TRUE;
		ELSE
			freshbar_col:= FALSE; (*ПОСТАВИТИ В ЗАЛЕЖНІСТЬ ВІД ЗОВНІШНЬОЇ ТЕМПЕРАТУРИ*)
		END_IF
	END_IF

	IF t_su > t_max THEN
		su_col_pidloga:=FALSE;
		su_col_stina:=FALSE;
			serverna_col:=FALSE;
	ELSE
		IF t_su< t_min THEN
			su_col_pidloga:=TRUE;
			su_col_stina:=TRUE;
			serverna_col:=TRUE;
		ELSE
			su_col_pidloga:=FALSE; (*ПОСТАВИТИ В ЗАЛЕЖНІСТЬ ВІД ЗОВНІШНЬОЇ ТЕМПЕРАТУРИ*)
			su_col_stina:=FALSE;
			serverna_col:=FALSE;
		END_IF
	END_IF

	IF t_spalnya>t_max THEN (*щоб не вистигала підлога*)
		spalnya_col:=FALSE;
	ELSE
		IF t_spalnya<t_min THEN
			spalnya_col:=TRUE;
		ELSE
			spalnya_col:=SPALNYA_HVAC.tepla_pidloga;
		END_IF
	END_IF


END_IF

(*

IF VITALNYA_HVAC.heat_mode=0 THEN
				VITALNYA_HVAC.fancoil_speed:=0;
				(*VITALNYA_HVAC.collector:=2#00000000; all closed*)
				VITALNYA_HVAC.klapan:=16#7FFF;(*full closed*)
				VITALNYA_HVAC.zaslinka:=TRUE;(*closed*)
	END_IF

	IF KINO_HVAC.heat_mode=0 THEN
				KINO_HVAC.fancoil_speed:=0;
				(*KINO_HVAC.collector:=2#00000000; all closed*)
				KINO_HVAC.klapan:=16#7FFF;(*full closed*)
				KINO_HVAC.zaslinka:=TRUE;(*closed*)
	END_IF

	IF STUDIO_HVAC.heat_mode=0 THEN
				STUDIO_HVAC.fancoil_speed:=0;
				(*STUDIO_HVAC.collector:=2#00000000; all closed*)
				STUDIO_HVAC.klapan:=16#7FFF;(*full closed*)
				STUDIO_HVAC.zaslinka:=TRUE;(*closed*)
	END_IF

	IF KABINET_HVAC.heat_mode=0 THEN
				KABINET_HVAC.fancoil_speed:=0;
				(*KABINET_HVAC.collector:=2#00000000; all closed*)
				KABINET_HVAC.klapan:=16#7FFF;(*full closed*)
				KABINET_HVAC.zaslinka:=TRUE;(*closed*)
	END_IF

	IF DYTJACHA_HVAC.heat_mode=0 THEN
				DYTJACHA_HVAC.fancoil_speed:=0;
				(*DYTJACHA_HVAC.collector:=2#00000000; all closed*)
				DYTJACHA_HVAC.klapan:=16#7FFF;(*full closed*)
				DYTJACHA_HVAC.zaslinka:=TRUE;(*closed*)
	END_IF

	IF SPALNYA_HVAC.heat_mode=0 THEN
				SPALNYA_HVAC.fancoil_speed:=0;
				(*SPALNYA_HVAC.collector:=2#00000000; all closed*)
				SPALNYA_HVAC.klapan:=16#7FFF;(*full closed*)
				SPALNYA_HVAC.zaslinka:=TRUE;(*closed*)
	END_IF
*)





(*локальні змінні для фенкойлів 3го поверхну об'явлені в області виходів*)

(*------------------------fancoil speed --------------------------------------------------*)
IF EIB.fb_vitalnya_damper_ctrl_rec.bData THEN
	vitalnya_hvac.fancoil_speed:=1;
ELSE
	IF vitalnya_HVAC.heating_signal = 0  THEN
		CASE vitalnya_hvac.fancoil_speed OF
			0:	IF vitalnya_hvac.cooling_signal>0 THEN vitalnya_HVAC.fancoil_speed:=1; END_IF

			1:	IF vitalnya_hvac.cooling_signal=0 THEN vitalnya_HVAC.fancoil_speed:=0; END_IF
				IF vitalnya_hvac.cooling_signal>50 THEN  vitalnya_HVAC.fancoil_speed:=2; END_IF

			2:	IF vitalnya_hvac.cooling_signal=0 THEN vitalnya_HVAC.fancoil_speed:=0; END_IF
				IF vitalnya_hvac.cooling_signal>75  THEN vitalnya_HVAC.fancoil_speed:=3; END_IF
				IF vitalnya_hvac.cooling_signal<45  THEN vitalnya_HVAC.fancoil_speed:=1; END_IF

			3:	IF vitalnya_hvac.cooling_signal=0 THEN vitalnya_HVAC.fancoil_speed:=0; END_IF
				IF vitalnya_hvac.cooling_signal<75  THEN vitalnya_HVAC.fancoil_speed:=2; END_IF
		END_CASE
	END_IF

	IF vitalnya_HVAC.cooling_signal = 0 THEN
		CASE vitalnya_hvac.fancoil_speed OF
			0:	IF vitalnya_hvac.heating_signal>0 THEN vitalnya_HVAC.fancoil_speed:=1; END_IF

			1:	IF vitalnya_hvac.heating_signal=0 THEN vitalnya_HVAC.fancoil_speed:=0; END_IF
				IF vitalnya_hvac.heating_signal>50 THEN  vitalnya_HVAC.fancoil_speed:=2; END_IF

			2:	IF vitalnya_hvac.heating_signal=0 THEN vitalnya_HVAC.fancoil_speed:=0; END_IF
				IF vitalnya_hvac.heating_signal>75  THEN vitalnya_HVAC.fancoil_speed:=3; END_IF
				IF vitalnya_hvac.heating_signal<45  THEN vitalnya_HVAC.fancoil_speed:=1; END_IF

			3:	IF vitalnya_hvac.heating_signal=0 THEN vitalnya_HVAC.fancoil_speed:=0; END_IF
				IF vitalnya_hvac.heating_signal<75  THEN vitalnya_HVAC.fancoil_speed:=2; END_IF
		END_CASE
	END_IF
END_IF

IF EIB.fb_kino_damper_ctrl_rec.bData THEN
	kino_hvac.fancoil_speed:=1;
ELSE
	IF kino_HVAC.heating_signal = 0 THEN
		CASE kino_hvac.fancoil_speed OF
			0:	IF kino_hvac.cooling_signal>0 THEN kino_HVAC.fancoil_speed:=1; END_IF

			1:	IF kino_hvac.cooling_signal=0 THEN kino_HVAC.fancoil_speed:=0; END_IF
				IF kino_hvac.cooling_signal>50 THEN  kino_HVAC.fancoil_speed:=2; END_IF

			2:	IF kino_hvac.cooling_signal=0 THEN kino_HVAC.fancoil_speed:=0; END_IF
				IF kino_hvac.cooling_signal>75  THEN kino_HVAC.fancoil_speed:=3; END_IF
				IF kino_hvac.cooling_signal<45  THEN kino_HVAC.fancoil_speed:=1; END_IF

			3:	IF kino_hvac.cooling_signal=0 THEN kino_HVAC.fancoil_speed:=0; END_IF
				IF kino_hvac.cooling_signal<75  THEN kino_HVAC.fancoil_speed:=2; END_IF
		END_CASE
	END_IF
	IF kino_HVAC.cooling_signal = 0 THEN
		CASE kino_hvac.fancoil_speed OF
			0:	IF kino_hvac.heating_signal>0 THEN kino_HVAC.fancoil_speed:=1; END_IF

			1:	IF kino_hvac.heating_signal=0 THEN kino_HVAC.fancoil_speed:=0; END_IF
				IF kino_hvac.heating_signal>50 THEN  kino_HVAC.fancoil_speed:=2; END_IF

			2:	IF kino_hvac.heating_signal=0 THEN kino_HVAC.fancoil_speed:=0; END_IF
				IF kino_hvac.heating_signal>75  THEN kino_HVAC.fancoil_speed:=3; END_IF
				IF kino_hvac.heating_signal<45  THEN kino_HVAC.fancoil_speed:=1; END_IF

			3:	IF kino_hvac.heating_signal=0 THEN kino_HVAC.fancoil_speed:=0; END_IF
				IF kino_hvac.heating_signal<75  THEN kino_HVAC.fancoil_speed:=2; END_IF
		END_CASE
	END_IF
END_IF

IF EIB.fb_kabinet_damper_ctrl_rec.bData THEN
	kabinet_hvac.fancoil_speed:=1;
ELSE
	IF kabinet_HVAC.heating_signal = 0 THEN
		CASE kabinet_hvac.fancoil_speed OF
			0:	IF kabinet_hvac.cooling_signal>0 THEN kabinet_HVAC.fancoil_speed:=1; END_IF

			1:	IF kabinet_hvac.cooling_signal=0 THEN kabinet_HVAC.fancoil_speed:=0; END_IF
				IF kabinet_hvac.cooling_signal>50 THEN  kabinet_HVAC.fancoil_speed:=2; END_IF

			2:	IF kabinet_hvac.cooling_signal=0 THEN kabinet_HVAC.fancoil_speed:=0; END_IF
				IF kabinet_hvac.cooling_signal>75  THEN kabinet_HVAC.fancoil_speed:=3; END_IF
				IF kabinet_hvac.cooling_signal<45  THEN kabinet_HVAC.fancoil_speed:=1; END_IF

			3:	IF kabinet_hvac.cooling_signal=0 THEN kabinet_HVAC.fancoil_speed:=0; END_IF
				IF kabinet_hvac.cooling_signal<75  THEN kabinet_HVAC.fancoil_speed:=2; END_IF
		END_CASE
	END_IF
	IF kabinet_HVAC.cooling_signal = 0 THEN
		CASE kabinet_hvac.fancoil_speed OF
			0:	IF kabinet_hvac.heating_signal>0 THEN kabinet_HVAC.fancoil_speed:=1; END_IF

			1:	IF kabinet_hvac.heating_signal=0 THEN kabinet_HVAC.fancoil_speed:=0; END_IF
				IF kabinet_hvac.heating_signal>50 THEN  kabinet_HVAC.fancoil_speed:=2; END_IF

			2:	IF kabinet_hvac.heating_signal=0 THEN kabinet_HVAC.fancoil_speed:=0; END_IF
				IF kabinet_hvac.heating_signal>75  THEN kabinet_HVAC.fancoil_speed:=3; END_IF
				IF kabinet_hvac.heating_signal<45  THEN kabinet_HVAC.fancoil_speed:=1; END_IF

			3:	IF kabinet_hvac.heating_signal=0 THEN kabinet_HVAC.fancoil_speed:=0; END_IF
				IF kabinet_hvac.heating_signal<75  THEN kabinet_HVAC.fancoil_speed:=2; END_IF
		END_CASE
	END_IF
END_IF

IF EIB.fb_dytjacha_damper_ctrl_rec.bData THEN
	dytjacha_hvac.fancoil_speed:=1;
ELSE
	IF dytjacha_HVAC.heating_signal = 0 THEN
		CASE dytjacha_hvac.fancoil_speed OF
			0:	IF dytjacha_hvac.cooling_signal>0 THEN dytjacha_HVAC.fancoil_speed:=1; END_IF

			1:	IF dytjacha_hvac.cooling_signal=0 THEN dytjacha_HVAC.fancoil_speed:=0; END_IF
				IF dytjacha_hvac.cooling_signal>50 THEN  dytjacha_HVAC.fancoil_speed:=2; END_IF

			2:	IF dytjacha_hvac.cooling_signal=0 THEN dytjacha_HVAC.fancoil_speed:=0; END_IF
				IF dytjacha_hvac.cooling_signal>75  THEN dytjacha_HVAC.fancoil_speed:=3; END_IF
				IF dytjacha_hvac.cooling_signal<45  THEN dytjacha_HVAC.fancoil_speed:=1; END_IF

			3:	IF dytjacha_hvac.cooling_signal=0 THEN dytjacha_HVAC.fancoil_speed:=0; END_IF
				IF dytjacha_hvac.cooling_signal<75  THEN dytjacha_HVAC.fancoil_speed:=2; END_IF
		END_CASE
	END_IF
	IF dytjacha_HVAC.cooling_signal = 0 THEN
		CASE dytjacha_hvac.fancoil_speed OF
			0:	IF dytjacha_hvac.heating_signal>0 THEN dytjacha_HVAC.fancoil_speed:=1; END_IF

			1:	IF dytjacha_hvac.heating_signal=0 THEN dytjacha_HVAC.fancoil_speed:=0; END_IF
				IF dytjacha_hvac.heating_signal>50 THEN  dytjacha_HVAC.fancoil_speed:=2; END_IF

			2:	IF dytjacha_hvac.heating_signal=0 THEN dytjacha_HVAC.fancoil_speed:=0; END_IF
				IF dytjacha_hvac.heating_signal>75  THEN dytjacha_HVAC.fancoil_speed:=3; END_IF
				IF dytjacha_hvac.heating_signal<45  THEN dytjacha_HVAC.fancoil_speed:=1; END_IF

			3:	IF dytjacha_hvac.heating_signal=0 THEN dytjacha_HVAC.fancoil_speed:=0; END_IF
				IF dytjacha_hvac.heating_signal<75  THEN dytjacha_HVAC.fancoil_speed:=2; END_IF
		END_CASE
	END_IF
END_IF

IF EIB.fb_spalnya_damper_ctrl_rec.bData THEN
	spalnya_hvac.fancoil_speed:=1;
ELSE
	IF spalnya_HVAC.heating_signal = 0 THEN
		CASE spalnya_hvac.fancoil_speed OF
			0:	IF spalnya_hvac.cooling_signal>0 THEN spalnya_HVAC.fancoil_speed:=1; END_IF

			1:	IF spalnya_hvac.cooling_signal=0 THEN spalnya_HVAC.fancoil_speed:=0; END_IF
				IF spalnya_hvac.cooling_signal>50 THEN  spalnya_HVAC.fancoil_speed:=2; END_IF

			2:	IF spalnya_hvac.cooling_signal=0 THEN spalnya_HVAC.fancoil_speed:=0; END_IF
				IF spalnya_hvac.cooling_signal>75  THEN spalnya_HVAC.fancoil_speed:=3; END_IF
				IF spalnya_hvac.cooling_signal<45  THEN spalnya_HVAC.fancoil_speed:=1; END_IF

			3:	IF spalnya_hvac.cooling_signal=0 THEN spalnya_HVAC.fancoil_speed:=0; END_IF
				IF spalnya_hvac.cooling_signal<75  THEN spalnya_HVAC.fancoil_speed:=2; END_IF
		END_CASE
	END_IF
	IF spalnya_HVAC.cooling_signal = 0 THEN
		CASE spalnya_hvac.fancoil_speed OF
			0:	IF spalnya_hvac.heating_signal>0 THEN spalnya_HVAC.fancoil_speed:=1; END_IF

			1:	IF spalnya_hvac.heating_signal=0 THEN spalnya_HVAC.fancoil_speed:=0; END_IF
				IF spalnya_hvac.heating_signal>50 THEN  spalnya_HVAC.fancoil_speed:=2; END_IF

			2:	IF spalnya_hvac.heating_signal=0 THEN spalnya_HVAC.fancoil_speed:=0; END_IF
				IF spalnya_hvac.heating_signal>75  THEN spalnya_HVAC.fancoil_speed:=3; END_IF
				IF spalnya_hvac.heating_signal<45  THEN spalnya_HVAC.fancoil_speed:=1; END_IF

			3:	IF spalnya_hvac.heating_signal=0 THEN spalnya_HVAC.fancoil_speed:=0; END_IF
				IF spalnya_hvac.heating_signal<75  THEN spalnya_HVAC.fancoil_speed:=2; END_IF
		END_CASE
	END_IF
END_IF
CASE DYTJACHA_HVAC.fancoil_speed OF
	0:	fancoil_dytjacha_low:=FALSE;
		fancoil_dytjacha_med:=FALSE;
		fancoil_dytjacha_high:=FALSE;

	1:	fancoil_dytjacha_low:=TRUE;
		fancoil_dytjacha_med:=FALSE;
		fancoil_dytjacha_high:=FALSE;

	2:	fancoil_dytjacha_low:=FALSE;
		fancoil_dytjacha_med:=TRUE;
		fancoil_dytjacha_high:=FALSE;

	3:	fancoil_dytjacha_low:=FALSE;
		fancoil_dytjacha_med:=FALSE;
		fancoil_dytjacha_high:=TRUE;
END_CASE

CASE SPALNYA_HVAC.fancoil_speed OF
	0:	fancoil_spalnya_low:=FALSE;
		fancoil_spalnya_med:=FALSE;
		fancoil_spalnya_high:=FALSE;

	1:	fancoil_spalnya_low:=TRUE;
		fancoil_spalnya_med:=FALSE;
		fancoil_spalnya_high:=FALSE;

	2:	fancoil_spalnya_low:=FALSE;
		fancoil_spalnya_med:=TRUE;
		fancoil_spalnya_high:=FALSE;

	3:	fancoil_spalnya_low:=FALSE;
		fancoil_spalnya_med:=FALSE;
		fancoil_spalnya_high:=TRUE;
END_CASE
CASE KABINET_HVAC.fancoil_speed OF
	0:	data2floor[0].0:=0; (*запис в масив даних, що відправляються на 2й поверх*)
		data2floor[0].1:=0;
		data2floor[0].2:=0;

	1:	data2floor[0].0:=1; (*запис в масив даних, що відправляються на 2й поверх*)
		data2floor[0].1:=0;
		data2floor[0].2:=0;

	2:	data2floor[0].0:=0; (*запис в масив даних, що відправляються на 2й поверх*)
		data2floor[0].1:=1;
		data2floor[0].2:=0;

	3:	data2floor[0].0:=0; (*запис в масив даних, що відправляються на 2й поверх*)
		data2floor[0].1:=0;
		data2floor[0].2:=1;
END_CASE

CASE KINO_HVAC.fancoil_speed OF
	0:	data2floor[0].3:=0; (*запис в масив даних, що відправляються на 2й поверх*)
		data2floor[0].4:=0;
		data2floor[0].5:=0;

	1:	data2floor[0].3:=1; (*запис в масив даних, що відправляються на 2й поверх*)
		data2floor[0].4:=0;
		data2floor[0].5:=0;

	2:	data2floor[0].3:=0; (*запис в масив даних, що відправляються на 2й поверх*)
		data2floor[0].4:=1;
		data2floor[0].5:=0;

	3:	data2floor[0].3:=0; (*запис в масив даних, що відправляються на 2й поверх*)
		data2floor[0].4:=0;
		data2floor[0].5:=1;
END_CASE

CASE VITALNYA_HVAC.fancoil_speed OF
	0:	data1floor[0].0:=0; (*запис в масив даних, що відправляються на 1й поверх*)
		data1floor[0].1:=0;
		data1floor[0].2:=0;

	1:	data1floor[0].0:=1; (*запис в масив даних, що відправляються на 1й поверх*)
		data1floor[0].1:=0;
		data1floor[0].2:=0;

	2:	data1floor[0].0:=0; (*запис в масив даних, що відправляються на 1й поверх*)
		data1floor[0].1:=1;
		data1floor[0].2:=0;

	3:	data1floor[0].0:=0; (*запис в масив даних, що відправляються на 1й поверх*)
		data1floor[0].1:=0;
		data1floor[0].2:=1;
END_CASE

(*--------------------------------------klapany--------------------------------------------*)
(*data1floor[2]:=WORD_TO_BYTE(VITALNYA_HVAC.klapan); data1floor[3]:=WORD_TO_BYTE(SHR(VITALNYA_HVAC.klapan,8));*)
klapan_vitalnya:=VITALNYA_HVAC.klapan;
klapan_spalnya:=SPALNYA_HVAC.klapan;
klapan_dytjacha:=DYTJACHA_HVAC.klapan;

data2floor[2]:=WORD_TO_BYTE(KABINET_HVAC.klapan); data2floor[3]:=WORD_TO_BYTE(SHR(KABINET_HVAC.klapan,8));
data2floor[4]:=WORD_TO_BYTE(KINO_HVAC.klapan); data2floor[5]:=WORD_TO_BYTE(SHR(KINO_HVAC.klapan,8));

(*------------------------------zaslinky------------------------------------*)
z_vitalnya:=VITALNYA_HVAC.zaslinka;
z_kabinet:=KABINET_HVAC.zaslinka;
z_kino:=KINO_HVAC.zaslinka;
z_dytjacha:=DYTJACHA_HVAC.zaslinka;
z_spalnya:=SPALNYA_HVAC.zaslinka;

(*-----------------------------tepla pidloga-------------------------------*)
data1floor[0].4:=VITALNYA_HVAC.tepla_pidloga;
data2floor[1].0:=KABINET_HVAC.tepla_pidloga;
data2floor[1].1:=KABINET_HVAC.tepla_pidloga;
data2floor[1].2:=STUDIO_HVAC.tepla_pidloga;
data2floor[1].3:=STUDIO_HVAC.tepla_pidloga;

dytjacha_col:=DYTJACHA_HVAC.tepla_pidloga;
spalnya_col:=SPALNYA_HVAC.tepla_pidloga;
END_PROGRAM

(* POU ADS_write, ST *)
PROGRAM ADS_write
VAR
	write_timeout: TIME;
	b_write1, b_write2: BOOL;
	write_ads1, write_ads2, write_ads4: ADSWRITE;

	timer1, timer2:TP;
	errorcounter1, errorcounter2, pack_c:CTU ;
	test_word: WORD;
	i2,j2,i1,j1, i4,j4: INT;
	data_changed: BOOL;
	try_again2, try_again1, try_again4: BOOL;
	timer4: TP;
	b_write4: BOOL;
	errorcounter4: CTU;
END_VAR
write_timeout:=t#3s;

timer2(PT:=write_timeout*2);
timer2.IN:=FALSE;



FOR 2i:=0 TO (SIZEOF(data2floor))-1 DO
	IF data2floor[i2]<>data2floor_prev[i2]  OR try_again2 THEN
		b_write2:=TRUE;
		EXIT;
	ELSE
		b_write2:=FALSE;
	END_IF
END_FOR


FOR i1:=0 TO (SIZEOF(data1floor))-1 DO
	IF data1floor[i1]<>data1floor_prev[i1]  OR try_again1 THEN
		b_write1:=TRUE;
		EXIT;
	ELSE
		b_write1:=FALSE;
	END_IF
END_FOR


FOR i4:=0 TO (SIZEOF(data_derevo))-1 DO
	IF data_derevo[i4]<>data_derevo[i4]  OR try_again4 THEN
		b_write4:=TRUE;
		EXIT;
	ELSE
		b_write4:=FALSE;
	END_IF
END_FOR



(*
IF write_ads2.BUSY THEN b_write2:=FALSE; END_IF

	write_ads2(
		NETID:=ads_adr2,
		PORT:=800,
		IDXGRP:=16#4020,
		IDXOFFS:=300,
		WRITE:=b_write2,
		TMOUT:=write_timeout,
		LEN:=SIZEOF(data2floor),
		SRCADDR:=ADR(data2floor));
write_ads2.WRITE:=FALSE;

IF write_ads2.ERR AND NOT timer2.Q THEN
	timer2.IN:=TRUE;
	try_again2:=TRUE;
ELSE try_again2:=FALSE;
END_IF


(*1floor*)
FOR i1:=0 TO (SIZEOF(data1floor))-1 DO
	IF data1floor[i1]<>data1floor_prev[i1] AND NOT timer1.Q THEN
		b_write1:=TRUE;
		EXIT;
	ELSE
		b_write1:=FALSE;
	END_IF
END_FOR

IF try_again1 AND NOT timer1.Q THEN
	b_write1:=TRUE;
	try_again1:=FALSE;
END_IF

errorcounter1(cu:=write_ads1.ERR);

IF write_ads1.BUSY THEN b_write1:=FALSE; END_IF

	write_ads1(
		NETID:=ads_adr1,
		PORT:=800,
		IDXGRP:=16#4020,
		IDXOFFS:=300,
		WRITE:=b_write1,
		TMOUT:=write_timeout,
		LEN:=SIZEOF(data1floor),
		SRCADDR:=ADR(data1floor));

IF write_ads1.ERR AND NOT timer1.Q THEN
	timer1.IN:=TRUE;
	try_again1:=TRUE;
END_IF
timer1(PT:=write_timeout);
timer1.IN:=FALSE;



(*derevo*)
FOR i4:=0 TO (SIZEOF(data_derevo))-1 DO
	IF data_derevo[i4]<>data_derevo_prev[i4] AND NOT timer4.Q THEN
		b_write4:=TRUE;
		EXIT;
	ELSE
		b_write4:=FALSE;
	END_IF
END_FOR

IF try_again4 AND NOT timer4.Q THEN
	b_write4:=TRUE;
	try_again4:=FALSE;
END_IF

errorcounter4(cu:=write_ads4.ERR);


IF write_ads4.BUSY THEN b_write4:=FALSE; END_IF

	write_ads4(
		NETID:=ads_adr4,
		PORT:=800,
		IDXGRP:=16#4020,
		IDXOFFS:=400,
		WRITE:=b_write4,
		TMOUT:=write_timeout,
		LEN:=SIZEOF(data_derevo),
		SRCADDR:=ADR(data_derevo));

IF write_ads4.ERR AND NOT timer4.Q THEN
	timer4.IN:=TRUE;
	try_again4:=TRUE;
END_IF
timer4(PT:=write_timeout);
timer4.IN:=FALSE;
*)

FOR j1:=0 TO (SIZEOF(data1floor))-1 DO
	data1floor_prev[j1]:=data1floor[j1];
END_FOR

FOR j:=0 TO (SIZEOF(data2floor))-1 DO
	data2floor_prev[j]:=data2floor[j];
END_FOR

FOR j4:=0 TO (SIZEOF(data_derevo))-1 DO
	data_derevo_prev[j4]:=data_derevo[j4];
END_FOR
END_PROGRAM

(* POU ADS_Communication, CFC *)
PROGRAM ADS_Communication
VAR

	fb_floor1ADSwrite: ADSWRITE;
	fb_floor2ADSwrite: ADSWRITE;
	fb_floor4ADSwrite: ADSWRITE;

	heartbeat:TP;
END_VAR
VAR (* helpers for the ST form of the networks *)
	_t99 : BOOL;
	_t96 : BOOL;
END_VAR
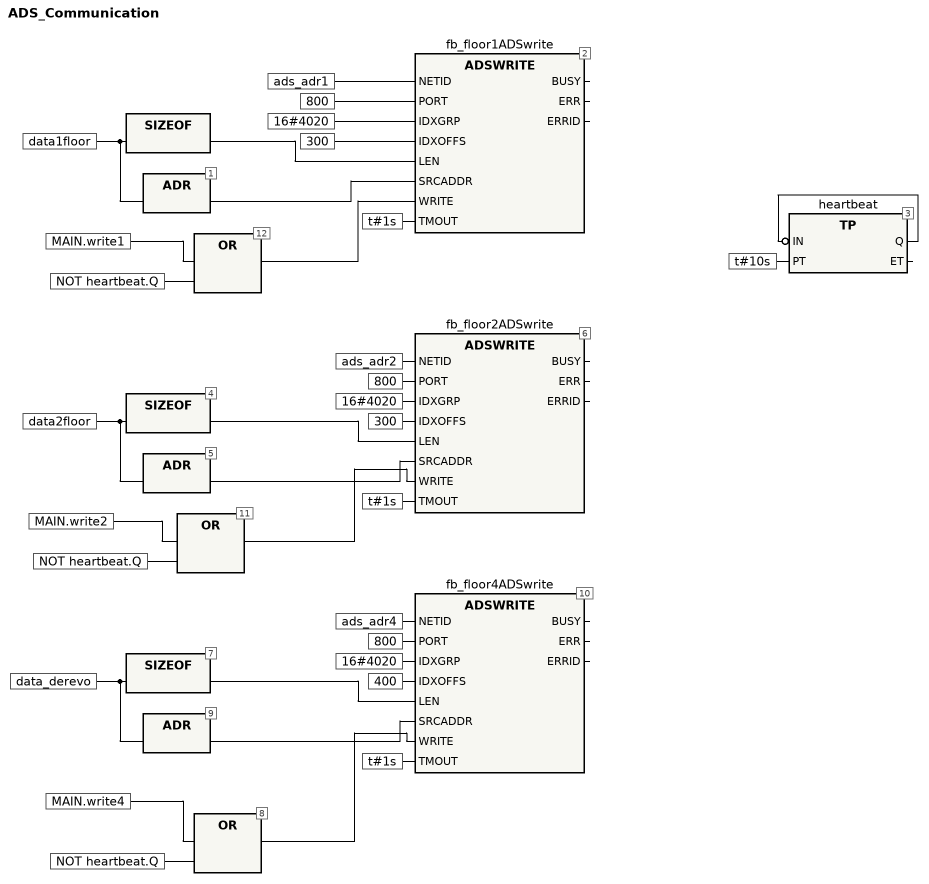
_CFC_ (* Continuous Function Chart, elements in execution order *)
#0 SIZEOF(data1floor)
#1 ADR(data1floor)
#2 fb_floor1ADSwrite:ADSWRITE(NETID: ads_adr1, PORT: 800, IDXGRP: 16#4020, IDXOFFS: 300, LEN: #0, SRCADDR: #1, WRITE: #12, TMOUT: t#1s)
#3 heartbeat:TP(IN: NOT #3.Q, PT: t#10s)
#4 SIZEOF(data2floor)
#5 ADR(data2floor)
#6 fb_floor2ADSwrite:ADSWRITE(NETID: ads_adr2, PORT: 800, IDXGRP: 16#4020, IDXOFFS: 300, LEN: #4, SRCADDR: #5, WRITE: #11, TMOUT: t#1s)
#7 SIZEOF(data_derevo)
#8 OR(MAIN.write4, NOT heartbeat.Q)
#9 ADR(data_derevo)
#10 fb_floor4ADSwrite:ADSWRITE(NETID: ads_adr4, PORT: 800, IDXGRP: 16#4020, IDXOFFS: 400, LEN: #7, SRCADDR: #9, WRITE: #8, TMOUT: t#1s)
#11 OR(MAIN.write2, NOT heartbeat.Q)
#12 OR(MAIN.write1, NOT heartbeat.Q)
_END_CFC_
(* the same logic as Structured Text *)
fb_floor1ADSwrite(NETID := ads_adr1, PORT := 800, IDXGRP := 16#4020, IDXOFFS := 300, LEN := SIZEOF(data1floor), SRCADDR := ADR(data1floor), WRITE := _t99, TMOUT := t#1s);
heartbeat(IN := NOT heartbeat.Q, PT := t#10s);
fb_floor2ADSwrite(NETID := ads_adr2, PORT := 800, IDXGRP := 16#4020, IDXOFFS := 300, LEN := SIZEOF(data2floor), SRCADDR := ADR(data2floor), WRITE := _t96, TMOUT := t#1s);
fb_floor4ADSwrite(NETID := ads_adr4, PORT := 800, IDXGRP := 16#4020, IDXOFFS := 400, LEN := SIZEOF(data_derevo), SRCADDR := ADR(data_derevo), WRITE := MAIN.write4 OR NOT heartbeat.Q, TMOUT := t#1s);
_t96 := MAIN.write2 OR NOT heartbeat.Q;
_t99 := MAIN.write1 OR NOT heartbeat.Q;
END_PROGRAM

(* POU HVAC/summer, ST *)
PROGRAM summer
VAR

END_VAR
data1floor[0].3:=heating_mode;

(*--------------------------VITALNYA---------------------------------------------------------------*)

	IF VITALNYA_HVAC.heat_mode=2 THEN (*heat*)
		IF heating_mode THEN VITALNYA_HVAC.zaslinka:=TRUE;(*closed*) ELSE VITALNYA_HVAC.zaslinka:=FALSE; (*opened*)END_IF;
		VITALNYA_HVAC.tepla_pidloga:=TRUE; (*all opened*);
		CASE VITALNYA_HVAC.heat_speed OF
			1:	VITALNYA_HVAC.fancoil_speed:=1;
				IF NOT heating_mode THEN  VITALNYA_HVAC.klapan:=16#0; ELSE VITALNYA_HVAC.klapan:=16#3FFF;END_IF
			2:	VITALNYA_HVAC.fancoil_speed:=2;
				IF NOT heating_mode THEN  VITALNYA_HVAC.klapan:=16#0; ELSE VITALNYA_HVAC.klapan:=16#5FFF;END_IF
			3:	VITALNYA_HVAC.fancoil_speed:=3;
				IF NOT heating_mode THEN  VITALNYA_HVAC.klapan:=16#0; ELSE VITALNYA_HVAC.klapan:=16#7FFF;END_IF
		END_CASE
	END_IF

	IF VITALNYA_HVAC.heat_mode=1 THEN (*cool*)
		IF  heating_mode THEN VITALNYA_HVAC.klapan:=16#0;(*full closed*) END_IF
		IF  heating_mode THEN VITALNYA_HVAC.zaslinka:=FALSE; ELSE VITALNYA_HVAC.zaslinka:=TRUE; END_IF
				VITALNYA_HVAC.tepla_pidloga:=FALSE; (*all closed*)

			CASE VITALNYA_HVAC.heat_speed OF
			1:	VITALNYA_HVAC.fancoil_speed:=1;
				IF NOT heating_mode THEN  VITALNYA_HVAC.klapan:=16#3FFF; ELSE VITALNYA_HVAC.klapan:=16#0;END_IF
			2:	VITALNYA_HVAC.fancoil_speed:=2;
				IF NOT heating_mode THEN  VITALNYA_HVAC.klapan:=16#5FFF; ELSE VITALNYA_HVAC.klapan:=16#0;END_IF
			3:	VITALNYA_HVAC.fancoil_speed:=3;
				IF NOT heating_mode THEN  VITALNYA_HVAC.klapan:=16#7FFF; ELSE VITALNYA_HVAC.klapan:=16#0;END_IF
		END_CASE
	END_IF

	IF VITALNYA_HVAC.heat_mode=3 THEN (*fan*)
		VITALNYA_HVAC.tepla_pidloga:=FALSE;

		CASE VITALNYA_HVAC.heat_speed OF
			1:	VITALNYA_HVAC.fancoil_speed:=0;
				VITALNYA_HVAC.zaslinka:=TRUE;(*closed*)
				VITALNYA_HVAC.klapan:=16#0;(*full closed*)
			2:	VITALNYA_HVAC.fancoil_speed:=2;
				VITALNYA_HVAC.zaslinka:=FALSE;(*opened*)
				VITALNYA_HVAC.klapan:=16#7FFF;
			3:	VITALNYA_HVAC.fancoil_speed:=3;
				VITALNYA_HVAC.zaslinka:=FALSE;(*opened*)
				VITALNYA_HVAC.klapan:=16#7FFF;
		END_CASE
	IF t_out<0 THEN VITALNYA_HVAC.klapan:=16#5FFF; ELSE VITALNYA_HVAC.klapan:=16#0;END_IF
	END_IF



(*--------------------------KABINET---------------------------------------------------------------*)
(*реверс двигуна клапана*)

	IF kabinet_HVAC.heat_mode=2 THEN (*heat*)
		IF heating_mode THEN kabinet_HVAC.zaslinka:=TRUE;(*closed*) ELSE kabinet_HVAC.zaslinka:=FALSE; (*opened*)END_IF;
		kabinet_HVAC.tepla_pidloga:=TRUE; (*all opened*);
		CASE kabinet_HVAC.heat_speed OF
			1:	kabinet_HVAC.fancoil_speed:=1;
				IF heating_mode THEN  kabinet_HVAC.klapan:=16#0; ELSE kabinet_HVAC.klapan:=16#7FFF;END_IF
			2:	kabinet_HVAC.fancoil_speed:=2;
				IF heating_mode THEN  kabinet_HVAC.klapan:=16#0; ELSE kabinet_HVAC.klapan:=16#5FFF;END_IF
			3:	kabinet_HVAC.fancoil_speed:=3;
				IF heating_mode THEN  kabinet_HVAC.klapan:=16#0; ELSE kabinet_HVAC.klapan:=16#3FFF;END_IF
		END_CASE
	END_IF

	IF kabinet_HVAC.heat_mode=1 THEN (*cool*)
		IF NOT heating_mode THEN kabinet_HVAC.klapan:=16#0;(*full closed*) END_IF
		IF NOT heating_mode THEN kabinet_HVAC.zaslinka:=FALSE; ELSE kabinet_HVAC.zaslinka:=TRUE; END_IF
				kabinet_HVAC.tepla_pidloga:=FALSE; (*all closed*)

			CASE kabinet_HVAC.heat_speed OF
			1:	kabinet_HVAC.fancoil_speed:=1;
				IF heating_mode THEN  kabinet_HVAC.klapan:=16#7FFF; ELSE kabinet_HVAC.klapan:=16#0;END_IF
			2:	kabinet_HVAC.fancoil_speed:=2;
				IF heating_mode THEN  kabinet_HVAC.klapan:=16#5FFF; ELSE kabinet_HVAC.klapan:=16#0;END_IF
			3:	kabinet_HVAC.fancoil_speed:=3;
				IF heating_mode THEN  kabinet_HVAC.klapan:=16#3FFF; ELSE kabinet_HVAC.klapan:=16#0;END_IF
		END_CASE
	END_IF

	IF kabinet_HVAC.heat_mode=3 THEN (*fan*)
		kabinet_HVAC.tepla_pidloga:=FALSE;
		IF t_out<0 THEN kabinet_HVAC.klapan:=16#3FFF;(*30%*) ELSE kabinet_HVAC.klapan:=16#0;END_IF
		CASE kabinet_HVAC.heat_speed OF
			1:	kabinet_HVAC.fancoil_speed:=0;
				kabinet_HVAC.zaslinka:=TRUE;(*closed*)
				kabinet_HVAC.klapan:=16#0;(*full closed*)
			2:	kabinet_HVAC.fancoil_speed:=2;
				kabinet_HVAC.zaslinka:=FALSE;(*opened*)
				kabinet_HVAC.klapan:=16#7FFF;
			3:	kabinet_HVAC.fancoil_speed:=3;
				kabinet_HVAC.zaslinka:=FALSE;(*opened*)
				kabinet_HVAC.klapan:=16#7FFF;
		END_CASE
	END_IF


(*--------------------------KINO---------------------------------------------------------------*)
(*реверс двигуна клапана*)

	IF KINO_HVAC.heat_mode=2 THEN (*heat*)
		IF heating_mode THEN KINO_HVAC.zaslinka:=TRUE;(*closed*) ELSE KINO_HVAC.zaslinka:=FALSE; (*opened*)END_IF;
		KINO_HVAC.tepla_pidloga:=TRUE; (*all opened*);
		CASE KINO_HVAC.heat_speed OF
			1:	KINO_HVAC.fancoil_speed:=1;
				IF NOT heating_mode THEN  KINO_HVAC.klapan:=16#0; ELSE KINO_HVAC.klapan:=16#5FFF;END_IF
			2:	KINO_HVAC.fancoil_speed:=2;
				IF NOT heating_mode THEN  KINO_HVAC.klapan:=16#0; ELSE KINO_HVAC.klapan:=16#3FFF;END_IF
			3:	KINO_HVAC.fancoil_speed:=3;
				IF NOT heating_mode THEN  KINO_HVAC.klapan:=16#0; ELSE KINO_HVAC.klapan:=16#0;END_IF
		END_CASE
	END_IF

	IF KINO_HVAC.heat_mode=1 THEN (*cool*)
		IF  heating_mode THEN KINO_HVAC.klapan:=16#7FFF;(*full closed*) END_IF
		IF  heating_mode THEN KINO_HVAC.zaslinka:=FALSE; ELSE KINO_HVAC.zaslinka:=TRUE; END_IF
				KINO_HVAC.tepla_pidloga:=FALSE; (*all closed*)

			CASE KINO_HVAC.heat_speed OF
			1:	KINO_HVAC.fancoil_speed:=1;
				IF NOT heating_mode THEN  KINO_HVAC.klapan:=16#5FFF; ELSE KINO_HVAC.klapan:=16#7FFF;END_IF
			2:	KINO_HVAC.fancoil_speed:=2;
				IF NOT heating_mode THEN  KINO_HVAC.klapan:=16#3FFF; ELSE KINO_HVAC.klapan:=16#7FFF;END_IF
			3:	KINO_HVAC.fancoil_speed:=3;
				IF NOT heating_mode THEN  KINO_HVAC.klapan:=16#0; ELSE KINO_HVAC.klapan:=16#7FFF;END_IF
		END_CASE
	END_IF

	IF KINO_HVAC.heat_mode=3 THEN (*fan*)
		KINO_HVAC.tepla_pidloga:=FALSE;

		CASE KINO_HVAC.heat_speed OF
			1:	KINO_HVAC.fancoil_speed:=0;
				KINO_HVAC.zaslinka:=TRUE;(*closed*)
				KINO_HVAC.klapan:=16#7FFF;(*full closed*)
			2:	KINO_HVAC.fancoil_speed:=2;
				KINO_HVAC.zaslinka:=FALSE;(*opened*)
				KINO_HVAC.klapan:=16#7FFF;
			3:	KINO_HVAC.fancoil_speed:=3;
				KINO_HVAC.zaslinka:=FALSE;(*opened*)
				KINO_HVAC.klapan:=16#7FFF;
		END_CASE
		IF t_out<0 THEN KINO_HVAC.klapan:=16#5FFF;  ELSE KINO_HVAC.klapan:=16#7FFF;END_IF
	END_IF

(*--------------------------DYTJACHA---------------------------------------------------------------*)
(*реверс двигуна клапана*)

	IF dytjacha_HVAC.heat_mode=2 THEN (*heat*)
		IF heating_mode THEN dytjacha_HVAC.zaslinka:=TRUE;(*closed*) ELSE dytjacha_HVAC.zaslinka:=FALSE; (*opened*)END_IF;
		dytjacha_HVAC.tepla_pidloga:=TRUE; (*all opened*);
		CASE dytjacha_HVAC.heat_speed OF
			1:	dytjacha_HVAC.fancoil_speed:=1;
				IF NOT heating_mode THEN  dytjacha_HVAC.klapan:=16#7FFF; ELSE dytjacha_HVAC.klapan:=16#5FFF;END_IF
			2:	dytjacha_HVAC.fancoil_speed:=2;
				IF NOT heating_mode THEN  dytjacha_HVAC.klapan:=16#7FFF; ELSE dytjacha_HVAC.klapan:=16#3FFF;END_IF
			3:	dytjacha_HVAC.fancoil_speed:=3;
				IF NOT heating_mode THEN  dytjacha_HVAC.klapan:=16#7FFF; ELSE dytjacha_HVAC.klapan:=16#0;END_IF
		END_CASE
	END_IF

	IF dytjacha_HVAC.heat_mode=1 THEN (*cool*)
		IF  heating_mode THEN dytjacha_HVAC.klapan:=16#7FFF;(*full closed*) END_IF
		IF  heating_mode THEN dytjacha_HVAC.zaslinka:=FALSE; ELSE dytjacha_HVAC.zaslinka:=TRUE; END_IF
				dytjacha_HVAC.tepla_pidloga:=FALSE; (*all closed*)

			CASE dytjacha_HVAC.heat_speed OF
			1:	dytjacha_HVAC.fancoil_speed:=1;
				IF heating_mode THEN  dytjacha_HVAC.klapan:=16#7FFF; ELSE dytjacha_HVAC.klapan:=16#0;END_IF
			2:	dytjacha_HVAC.fancoil_speed:=2;
				IF heating_mode THEN  dytjacha_HVAC.klapan:=16#5FFF; ELSE dytjacha_HVAC.klapan:=16#0;END_IF
			3:	dytjacha_HVAC.fancoil_speed:=3;
				IF heating_mode THEN  dytjacha_HVAC.klapan:=16#3FFF; ELSE dytjacha_HVAC.klapan:=16#0;END_IF
		END_CASE
	END_IF

	IF dytjacha_HVAC.heat_mode=3 THEN (*fan*)
		dytjacha_HVAC.tepla_pidloga:=FALSE;
		CASE dytjacha_HVAC.heat_speed OF
			1:	dytjacha_HVAC.fancoil_speed:=0;
				dytjacha_HVAC.zaslinka:=TRUE;(*closed*)
				dytjacha_HVAC.klapan:=16#0;(*full closed*)
			2:	dytjacha_HVAC.fancoil_speed:=2;
				dytjacha_HVAC.zaslinka:=FALSE;(*opened*)
				dytjacha_HVAC.klapan:=16#7FFF;
			3:	dytjacha_HVAC.fancoil_speed:=3;
				dytjacha_HVAC.zaslinka:=FALSE;(*opened*)
				dytjacha_HVAC.klapan:=16#7FFF;
		END_CASE
		IF t_out<0 THEN dytjacha_HVAC.klapan:=16#5FFF; ELSE dytjacha_HVAC.klapan:=16#7FFF;END_IF
	END_IF
(*--------------------------SPALNYA---------------------------------------------------------------*)

	IF SPALNYA_HVAC.heat_mode=2 THEN (*heat*)
		IF heating_mode THEN SPALNYA_HVAC.zaslinka:=TRUE;(*closed*) ELSE SPALNYA_HVAC.zaslinka:=FALSE; (*opened*)END_IF;
		SPALNYA_HVAC.tepla_pidloga:=TRUE; (*all opened*);
		CASE SPALNYA_HVAC.heat_speed OF
			1:	SPALNYA_HVAC.fancoil_speed:=1;
				IF NOT  heating_mode THEN  SPALNYA_HVAC.klapan:=16#0; ELSE SPALNYA_HVAC.klapan:=16#3FFF;END_IF
			2:	SPALNYA_HVAC.fancoil_speed:=2;
				IF NOT heating_mode THEN  SPALNYA_HVAC.klapan:=16#0; ELSE SPALNYA_HVAC.klapan:=16#5FFF;END_IF
			3:	SPALNYA_HVAC.fancoil_speed:=3;
				IF NOT heating_mode THEN  SPALNYA_HVAC.klapan:=16#0; ELSE SPALNYA_HVAC.klapan:=16#7FFF;END_IF
		END_CASE
	END_IF

	IF SPALNYA_HVAC.heat_mode=1 THEN (*cool*)
		IF  heating_mode THEN SPALNYA_HVAC.klapan:=16#5FFF;(*full closed*) END_IF
		IF  heating_mode THEN SPALNYA_HVAC.zaslinka:=FALSE; ELSE SPALNYA_HVAC.zaslinka:=TRUE; END_IF
				SPALNYA_HVAC.tepla_pidloga:=FALSE; (*all closed*)

			CASE SPALNYA_HVAC.heat_speed OF
			1:	SPALNYA_HVAC.fancoil_speed:=1;
				IF NOT heating_mode THEN  SPALNYA_HVAC.klapan:=16#3FFF; ELSE SPALNYA_HVAC.klapan:=16#0;END_IF
			2:	SPALNYA_HVAC.fancoil_speed:=2;
				IF NOT heating_mode THEN  SPALNYA_HVAC.klapan:=16#5FFF; ELSE SPALNYA_HVAC.klapan:=16#0;END_IF
			3:	SPALNYA_HVAC.fancoil_speed:=3;
				IF NOT heating_mode THEN  SPALNYA_HVAC.klapan:=16#7FFF; ELSE SPALNYA_HVAC.klapan:=16#0;END_IF
		END_CASE
	END_IF

	IF SPALNYA_HVAC.heat_mode=3 THEN (*fan*)
		SPALNYA_HVAC.tepla_pidloga:=FALSE;
		CASE SPALNYA_HVAC.heat_speed OF
			1:	SPALNYA_HVAC.fancoil_speed:=0;
				SPALNYA_HVAC.zaslinka:=TRUE;(*closed*)
				SPALNYA_HVAC.klapan:=16#0;(*full closed*)
			2:	SPALNYA_HVAC.fancoil_speed:=2;
				SPALNYA_HVAC.zaslinka:=FALSE;(*opened*)
				SPALNYA_HVAC.klapan:=16#0;
			3:	SPALNYA_HVAC.fancoil_speed:=3;
				SPALNYA_HVAC.zaslinka:=FALSE;(*opened*)
				SPALNYA_HVAC.klapan:=16#0;
		END_CASE
		IF t_out<0 THEN SPALNYA_HVAC.klapan:=16#3FFF;(*30%*) ELSE SPALNYA_HVAC.klapan:=16#0;END_IF
	END_IF
END_PROGRAM

(* POU HVAC/winter, ST *)
PROGRAM winter
VAR

END_VAR
(*1-COOL mode 2-HEAT mode, 3-FAN mode*)

(*--------------------------VITALNYA---------------------------------------------------------------*)

	IF VITALNYA_HVAC.heat_mode=2 THEN
				VITALNYA_HVAC.zaslinka:=TRUE;(*closed*)
				VITALNYA_HVAC.tepla_pidloga:=TRUE; (*all opened*)
		CASE VITALNYA_HVAC.heat_speed OF

			1:	VITALNYA_HVAC.fancoil_speed:=1;
				VITALNYA_HVAC.klapan:=16#3FFF;
			2:	VITALNYA_HVAC.fancoil_speed:=2;
				VITALNYA_HVAC.klapan:=16#5FFF;
			3:	VITALNYA_HVAC.fancoil_speed:=3;
				VITALNYA_HVAC.klapan:=16#7FFF;
		END_CASE
	END_IF

	IF VITALNYA_HVAC.heat_mode=1 THEN
				VITALNYA_HVAC.klapan:=16#0;(*full closed*)
				VITALNYA_HVAC.zaslinka:=FALSE;
				VITALNYA_HVAC.tepla_pidloga:=FALSE; (*all closed*)

			CASE VITALNYA_HVAC.heat_speed OF
			1:	VITALNYA_HVAC.fancoil_speed:=1;
			2:	VITALNYA_HVAC.fancoil_speed:=2;
			3:	VITALNYA_HVAC.fancoil_speed:=3;
		END_CASE
	END_IF

	IF VITALNYA_HVAC.heat_mode=3 THEN
		VITALNYA_HVAC.tepla_pidloga:=FALSE;
		IF t_out<0 THEN VITALNYA_HVAC.klapan:=16#3FFF;(*30%*) ELSE VITALNYA_HVAC.klapan:=16#0;END_IF
		CASE VITALNYA_HVAC.heat_speed OF
			1:	VITALNYA_HVAC.fancoil_speed:=0;
				VITALNYA_HVAC.zaslinka:=TRUE;(*closed*)
				VITALNYA_HVAC.klapan:=16#0;(*full closed*)
			2:	VITALNYA_HVAC.fancoil_speed:=2;
				VITALNYA_HVAC.zaslinka:=FALSE;(*opened*)
			3:	VITALNYA_HVAC.fancoil_speed:=3;
				VITALNYA_HVAC.zaslinka:=FALSE;(*opened*)
		END_CASE
	END_IF



(*--------------------------KABINET---------------------------------------------------------------*)
(*реверс двигуна клапана*)

	IF KABINET_HVAC.heat_mode=2 THEN
				KABINET_HVAC.zaslinka:=TRUE;(*closed*)
				KABINET_HVAC.tepla_pidloga:=TRUE; (*all opened*)
		CASE KABINET_HVAC.heat_speed OF

			1:	KABINET_HVAC.fancoil_speed:=1;
				KABINET_HVAC.klapan:=16#5FFF;
			2:	KABINET_HVAC.fancoil_speed:=2;
				KABINET_HVAC.klapan:=16#3FFF;
			3:	KABINET_HVAC.fancoil_speed:=3;
				KABINET_HVAC.klapan:=16#1FFF;
		END_CASE
	END_IF

	IF KABINET_HVAC.heat_mode=1 THEN
				KABINET_HVAC.klapan:=16#7FFF;(*full closed*)
				KABINET_HVAC.zaslinka:=FALSE;
				KABINET_HVAC.tepla_pidloga:=FALSE; (*all closed*)

			CASE KABINET_HVAC.heat_speed OF
			1:	KABINET_HVAC.fancoil_speed:=1;
			2:	KABINET_HVAC.fancoil_speed:=2;
			3:	KABINET_HVAC.fancoil_speed:=3;
		END_CASE
	END_IF

	IF KABINET_HVAC.heat_mode=3 THEN
		KABINET_HVAC.tepla_pidloga:=FALSE;
		IF t_out<0 THEN KABINET_HVAC.klapan:=16#5FFF;(*30%*) ELSE KABINET_HVAC.klapan:=16#7FFF;END_IF
		CASE KABINET_HVAC.heat_speed OF
			1:	KABINET_HVAC.fancoil_speed:=0;
				KABINET_HVAC.zaslinka:=TRUE;(*closed*)
				KABINET_HVAC.klapan:=16#7FFF;(*full closed*)
			2:	KABINET_HVAC.fancoil_speed:=2;
				KABINET_HVAC.zaslinka:=FALSE;(*opened*)
			3:	KABINET_HVAC.fancoil_speed:=3;
				KABINET_HVAC.zaslinka:=FALSE;(*opened*)
		END_CASE
	END_IF



(*--------------------------KINO---------------------------------------------------------------*)
(*реверс двигуна клапана*)
	IF KINO_HVAC.heat_mode=2 THEN
				KINO_HVAC.zaslinka:=TRUE;(*closed*)
				KINO_HVAC.tepla_pidloga:=TRUE; (*all opened*)
		CASE KINO_HVAC.heat_speed OF

			1:	KINO_HVAC.fancoil_speed:=1;
				KINO_HVAC.klapan:=16#5FFF;
			2:	KINO_HVAC.fancoil_speed:=2;
				KINO_HVAC.klapan:=16#3FFF;
			3:	KINO_HVAC.fancoil_speed:=3;
				KINO_HVAC.klapan:=16#1FFF;
		END_CASE
	END_IF

	IF KINO_HVAC.heat_mode=1 THEN
				KINO_HVAC.klapan:=16#0;(*full closed*)
				KINO_HVAC.zaslinka:=FALSE;
				KINO_HVAC.tepla_pidloga:=FALSE; (*all closed*)

			CASE KINO_HVAC.heat_speed OF
			1:	KINO_HVAC.fancoil_speed:=1;
			2:	KINO_HVAC.fancoil_speed:=2;
			3:	KINO_HVAC.fancoil_speed:=3;
		END_CASE
	END_IF

	IF KINO_HVAC.heat_mode=3 THEN
		KINO_HVAC.tepla_pidloga:=FALSE;
		IF t_out<0 THEN KINO_HVAC.klapan:=16#5FFF;(*30%*) ELSE KINO_HVAC.klapan:=16#7FFF;END_IF
		CASE KINO_HVAC.heat_speed OF
			1:	KINO_HVAC.fancoil_speed:=0;
				KINO_HVAC.zaslinka:=TRUE;(*closed*)
				KINO_HVAC.klapan:=16#7FFF;(*full closed*)
			2:	KINO_HVAC.fancoil_speed:=2;
				KINO_HVAC.zaslinka:=FALSE;(*opened*)
			3:	KINO_HVAC.fancoil_speed:=3;
				KINO_HVAC.zaslinka:=FALSE;(*opened*)
		END_CASE
	END_IF



(*--------------------------DYTJACHA---------------------------------------------------------------*)
(*реверс двигуна клапана*)
	IF DYTJACHA_HVAC.heat_mode=2 THEN
				DYTJACHA_HVAC.zaslinka:=TRUE;(*closed*)
				DYTJACHA_HVAC.tepla_pidloga:=TRUE; (*all opened*)
		CASE DYTJACHA_HVAC.heat_speed OF

			1:	DYTJACHA_HVAC.fancoil_speed:=1;
				DYTJACHA_HVAC.klapan:=16#5FFF;
			2:	DYTJACHA_HVAC.fancoil_speed:=2;
				DYTJACHA_HVAC.klapan:=16#3FFF;
			3:	DYTJACHA_HVAC.fancoil_speed:=3;
				DYTJACHA_HVAC.klapan:=16#1FFF;
		END_CASE
	END_IF

	IF DYTJACHA_HVAC.heat_mode=1 THEN
				DYTJACHA_HVAC.klapan:=16#7FFF;(*full closed*)
				DYTJACHA_HVAC.zaslinka:=FALSE;
				DYTJACHA_HVAC.tepla_pidloga:=FALSE; (*all closed*)

			CASE DYTJACHA_HVAC.heat_speed OF
			1:	DYTJACHA_HVAC.fancoil_speed:=1;
			2:	DYTJACHA_HVAC.fancoil_speed:=2;
			3:	DYTJACHA_HVAC.fancoil_speed:=3;
		END_CASE
	END_IF

	IF DYTJACHA_HVAC.heat_mode=3 THEN
		DYTJACHA_HVAC.tepla_pidloga:=FALSE;
		IF t_out<0 THEN DYTJACHA_HVAC.klapan:=16#5FFF;(*30%*) ELSE DYTJACHA_HVAC.klapan:=16#7FFF;END_IF
		CASE DYTJACHA_HVAC.heat_speed OF
			1:	DYTJACHA_HVAC.fancoil_speed:=0;
				DYTJACHA_HVAC.zaslinka:=TRUE;(*closed*)
				DYTJACHA_HVAC.klapan:=16#7FFF;(*full closed*)
			2:	DYTJACHA_HVAC.fancoil_speed:=2;
				DYTJACHA_HVAC.zaslinka:=FALSE;(*opened*)
			3:	DYTJACHA_HVAC.fancoil_speed:=3;
				DYTJACHA_HVAC.zaslinka:=FALSE;(*opened*)
		END_CASE
	END_IF



(*--------------------------SPALNYA---------------------------------------------------------------*)

	IF SPALNYA_HVAC.heat_mode=2 THEN
				SPALNYA_HVAC.zaslinka:=TRUE;(*closed*)
				SPALNYA_HVAC.tepla_pidloga:=TRUE; (*all opened*)
		CASE SPALNYA_HVAC.heat_speed OF

			1:	SPALNYA_HVAC.fancoil_speed:=1;
				SPALNYA_HVAC.klapan:=16#3FFF;
			2:	SPALNYA_HVAC.fancoil_speed:=2;
				SPALNYA_HVAC.klapan:=16#5FFF;
			3:	SPALNYA_HVAC.fancoil_speed:=3;
				SPALNYA_HVAC.klapan:=16#7FFF;
		END_CASE
	END_IF

	IF SPALNYA_HVAC.heat_mode=1 THEN
				SPALNYA_HVAC.klapan:=16#0;(*full closed*)
				SPALNYA_HVAC.zaslinka:=FALSE;
				SPALNYA_HVAC.tepla_pidloga:=FALSE; (*all closed*)

			CASE SPALNYA_HVAC.heat_speed OF
			1:	SPALNYA_HVAC.fancoil_speed:=1;
			2:	SPALNYA_HVAC.fancoil_speed:=2;
			3:	SPALNYA_HVAC.fancoil_speed:=3;
		END_CASE
	END_IF

	IF SPALNYA_HVAC.heat_mode=3 THEN
		SPALNYA_HVAC.tepla_pidloga:=FALSE;
		IF t_out<0 THEN SPALNYA_HVAC.klapan:=16#3FFF;(*30%*) ELSE SPALNYA_HVAC.klapan:=16#0;END_IF
		CASE SPALNYA_HVAC.heat_speed OF
			1:	SPALNYA_HVAC.fancoil_speed:=0;
				SPALNYA_HVAC.zaslinka:=TRUE;(*closed*)
				SPALNYA_HVAC.klapan:=16#0;(*full closed*)
			2:	SPALNYA_HVAC.fancoil_speed:=2;
				SPALNYA_HVAC.zaslinka:=FALSE;(*opened*)
			3:	SPALNYA_HVAC.fancoil_speed:=3;
				SPALNYA_HVAC.zaslinka:=FALSE;(*opened*)
		END_CASE
	END_IF
END_PROGRAM
